// TwinCAT 3 PLC project CassetteLoaderPLC
// ProgramVersion: 3.1.4024.0
// libraries:
//   SPT Base Types, * (Beckhoff Automation LLC)
//   SPT Components, * (Beckhoff Automation LLC)
//   SPT Event Logger, * (Beckhoff Automation LLC)
//   SPT Motion Control, * (Beckhoff Automation LLC)
//   SPT Utilities, * (Beckhoff Automation LLC)
//   Tc2_EtherCAT, * (Beckhoff Automation GmbH)
//   Tc2_Standard, * (Beckhoff Automation GmbH)
//   Tc2_System, * (Beckhoff Automation GmbH)
//   Tc3_EventLogger, * (Beckhoff Automation GmbH)
//   Tc3_Module, * (Beckhoff Automation GmbH)
//   Tc3_PackML_V2, * (Beckhoff Automation GmbH)
//   VisuDialogs, * (System)
//   VisuSymbols, * (System)
// project tree:
//   DUTs/Recipes/ ST_ElevatorRecipe.TcDUT, ST_LoaderRecipe.TcDUT, ST_ShuttleRecipe.TcDUT
//   DUTs/ ST_CassetteStatus.TcDUT, ST_PackML_Control.TcDUT, ST_PackML_Control_Simplified.TcDUT (not stored)
//   / GlobalTextList.TcGTLO, PlcTask.TcTTO, Visualization Manager.TcVMO (not stored)
//   Machine/EquipmentModules/ FB_CassetteLoader.TcPOU
//   Machine/ FB_Machine.TcPOU
//   Machine/HMI Connections/ FB_ControlSource_HMI.TcPOU, FB_ControlSource_HMI_Machine.TcPOU
//   Machine/Templates/ FB_EquipmentModuleTemplate.TcPOU
//   POUs/ MAIN.TcPOU
//   VISUs/VisuOjects/ V_MachineModule.TcVIS, V_Module.TcVIS
//   VISUs/ V_Main.TcVIS
// real-time tasks:
//   TASK PlcTask: cycle T#10ms, priority 20, ADS port 350
// motion (NC):
//   TASK NC-Task 1 SAF: cycle T#2ms, priority 4, ADS port 501
//   TASK NC-Task 1 SVB: cycle T#10ms, priority 8, ADS port 511
//   AXIS Axis-CassetteA (id 1)
//     Dynamic: Acceleration=607.875, Deceleration=607.875, Jerk=1823.62
//     Velo: RefSearch=4.0525, RefSync=4.0525, SlowManual=5, FastManual=50, Fast=405.25, Maximum=405.25
//     OtherSettings: AllowMotionCmdToSlave=true
//     encoder EncType=19
//       EncPara: ScaleFactorNumerator=5, ScaleFactorDenominator=1048576, MaxCount=#xffffffff
//     drive DrvType=16
//       DrvPara: MaxCount=#xffffffff, DriveControlDWord=#x00020000
//         Analog: VeloReferenz=445.775, VeloScale=32, TorqueSetpointScale=10, ScaleFactorActTorque=0.1
//         TimeComp: TaskDelayCycles=1
//     controller CtrType=1
//       CtrPara: PriorControlFactor=1
//         Observer: BandWidth=20
//   AXIS Axis-CassetteB (id 2)
//     Dynamic: Acceleration=607.875, Deceleration=607.875, Jerk=1823.62
//     Velo: RefSearch=4.0525, RefSync=4.0525, SlowManual=5, FastManual=50, Fast=405.25, Maximum=405.25
//     OtherSettings: AllowMotionCmdToSlave=true
//     encoder EncType=19
//       EncPara: ScaleFactorNumerator=5, ScaleFactorDenominator=1048576, MaxCount=#xffffffff
//     drive DrvType=16
//       DrvPara: MaxCount=#xffffffff, DriveControlDWord=#x00020000
//         Analog: VeloReferenz=445.775, VeloScale=32, TorqueSetpointScale=10, ScaleFactorActTorque=0.1
//         TimeComp: TaskDelayCycles=1
//     controller CtrType=1
//       CtrPara: PriorControlFactor=1
//         Observer: BandWidth=20
//   AXIS Axis-Shuttle (id 3)
//     Dynamic: Acceleration=607.875, Deceleration=607.875, Jerk=1823.62
//     Velo: RefSearch=4.0525, RefSync=4.0525, SlowManual=5, FastManual=50, Fast=405.25, Maximum=405.25
//     OtherSettings: AllowMotionCmdToSlave=true
//     encoder EncType=19
//       EncPara: ScaleFactorNumerator=5, ScaleFactorDenominator=1048576, MaxCount=#xffffffff
//     drive DrvType=16
//       DrvPara: MaxCount=#xffffffff, DriveControlDWord=#x00020000
//         Analog: VeloReferenz=445.775, VeloScale=32, TorqueSetpointScale=10, ScaleFactorActTorque=0.1
//         TimeComp: TaskDelayCycles=1
//     controller CtrType=1
//       CtrPara: PriorControlFactor=1
//         Observer: BandWidth=20
// I/O:
//   DEVICE Device 2 (EtherCAT), AmsNetId 169.254.242.100.3.1
//     Term 1 (EK1100) [EK1100 EtherCAT Coupler (2A E-Bus)]
//       Term 2 (EL1098) [EL1098 8Ch. Dig. Input 24V, 10µs, negative]
//       Term 3 (EL7201-9014) [EL7201-9014 1Ch. MDP742 Servo motor output stage with OCT (50V, 2.8A RMS) and STO input]
//       Term 4 (EL7201-9014) [EL7201-9014 1Ch. MDP742 Servo motor output stage with OCT (50V, 2.8A RMS) and STO input]
//       Term 5 (EL7201-9014) [EL7201-9014 1Ch. MDP742 Servo motor output stage with OCT (50V, 2.8A RMS) and STO input]
//       Term 6 (EL2904) [EL2904, 4 Ch. Safety Output 24V, 0.5A, TwinSAFE]
//         modules: Module 1 (FSOES), Module 2 (DO)
//       Term 7 (EL1918) [EL1918, 8Ch. Safety Input 24V, TwinSAFE]
//         modules: Module 1 (FSOE), Module 2 (FSLOGIC)
//       Term 8 (EL9011) [EL9011 End Terminal]
// variable links:
//   NC-Task 1 SAF/Axes/Axis-CassetteA <-> Device 2 (EtherCAT)/Term 1 (EK1100)/Term 3 (EL7201-9014)
//     Drive/Inputs/In/nDcOutputTime <-> InfoData/DcOutputShift
//     Drive/Inputs/In/nState1 <-> DRV Statusword/Statusword
//     Drive/Inputs/In/nState2 <-> DRV Statusword/Statusword @bit 8
//     Drive/Inputs/In/nState4 @bit 1 <-> WcState/InputToggle
//     Drive/Inputs/In/nState4 <-> WcState/WcState
//     Drive/Outputs/Out/nCtrl1 <-> DRV Controlword/Controlword
//     Drive/Outputs/Out/nCtrl2 <-> DRV Controlword/Controlword @bit 8
//     Drive/Outputs/Out/nDataOut2 <-> DRV Target velocity/Target velocity
//     Enc/Inputs/In/nDataIn1 <-> FB Position/Position
//     Enc/Inputs/In/nDcInputTime <-> InfoData/DcInputShift
//     Enc/Inputs/In/nState4 @bit 1 <-> WcState/InputToggle
//     Enc/Inputs/In/nState4 <-> WcState/WcState
//   NC-Task 1 SAF/Axes/Axis-CassetteB <-> Device 2 (EtherCAT)/Term 1 (EK1100)/Term 4 (EL7201-9014)
//     Drive/Inputs/In/nDcOutputTime <-> InfoData/DcOutputShift
//     Drive/Inputs/In/nState1 <-> DRV Statusword/Statusword
//     Drive/Inputs/In/nState2 <-> DRV Statusword/Statusword @bit 8
//     Drive/Inputs/In/nState4 @bit 1 <-> WcState/InputToggle
//     Drive/Inputs/In/nState4 <-> WcState/WcState
//     Drive/Outputs/Out/nCtrl1 <-> DRV Controlword/Controlword
//     Drive/Outputs/Out/nCtrl2 <-> DRV Controlword/Controlword @bit 8
//     Drive/Outputs/Out/nDataOut2 <-> DRV Target velocity/Target velocity
//     Enc/Inputs/In/nDataIn1 <-> FB Position/Position
//     Enc/Inputs/In/nDcInputTime <-> InfoData/DcInputShift
//     Enc/Inputs/In/nState4 @bit 1 <-> WcState/InputToggle
//     Enc/Inputs/In/nState4 <-> WcState/WcState
//   NC-Task 1 SAF/Axes/Axis-Shuttle <-> Device 2 (EtherCAT)/Term 1 (EK1100)/Term 5 (EL7201-9014)
//     Drive/Inputs/In/nDcOutputTime <-> InfoData/DcOutputShift
//     Drive/Inputs/In/nState1 <-> DRV Statusword/Statusword
//     Drive/Inputs/In/nState2 <-> DRV Statusword/Statusword @bit 8
//     Drive/Inputs/In/nState4 @bit 1 <-> WcState/InputToggle
//     Drive/Inputs/In/nState4 <-> WcState/WcState
//     Drive/Outputs/Out/nCtrl1 <-> DRV Controlword/Controlword
//     Drive/Outputs/Out/nCtrl2 <-> DRV Controlword/Controlword @bit 8
//     Drive/Outputs/Out/nDataOut2 <-> DRV Target velocity/Target velocity
//     Enc/Inputs/In/nDataIn1 <-> FB Position/Position
//     Enc/Inputs/In/nDcInputTime <-> InfoData/DcInputShift
//     Enc/Inputs/In/nState4 @bit 1 <-> WcState/InputToggle
//     Enc/Inputs/In/nState4 <-> WcState/WcState
//   CassetteLoaderPLC/CassetteLoaderPLC Instance <-> NC-Task 1 SAF/Axes/Axis-CassetteA
//     PlcTask Inputs/MAIN.CassetteLoaderMachine.CassetteLoaderEM.ElevatorAxisA.BasicAxis._Axis.NcToPlc <-> Outputs/ToPlc
//     PlcTask Outputs/MAIN.CassetteLoaderMachine.CassetteLoaderEM.ElevatorAxisA.BasicAxis._Axis.PlcToNc <-> Inputs/FromPlc
//   CassetteLoaderPLC/CassetteLoaderPLC Instance <-> NC-Task 1 SAF/Axes/Axis-CassetteB
//     PlcTask Inputs/MAIN.CassetteLoaderMachine.CassetteLoaderEM.ElevatorAxisB.BasicAxis._Axis.NcToPlc <-> Outputs/ToPlc
//     PlcTask Outputs/MAIN.CassetteLoaderMachine.CassetteLoaderEM.ElevatorAxisB.BasicAxis._Axis.PlcToNc <-> Inputs/FromPlc
//   CassetteLoaderPLC/CassetteLoaderPLC Instance <-> NC-Task 1 SAF/Axes/Axis-Shuttle
//     PlcTask Inputs/MAIN.CassetteLoaderMachine.CassetteLoaderEM.ShuttleAxis.BasicAxis._Axis.NcToPlc <-> Outputs/ToPlc
//     PlcTask Outputs/MAIN.CassetteLoaderMachine.CassetteLoaderEM.ShuttleAxis.BasicAxis._Axis.PlcToNc <-> Inputs/FromPlc

CONFIGURATION CassetteLoaderPLC
    RESOURCE PLC ON TwinCAT3
        TASK PlcTask(INTERVAL := T#10ms, PRIORITY := 20);
        PROGRAM MAIN WITH PlcTask : MAIN;
    END_RESOURCE
END_CONFIGURATION

// ---- DUTs/Recipes/ST_ElevatorRecipe.TcDUT
TYPE ST_ElevatorRecipe :
STRUCT
	    Velocity     : LREAL;
        Acceleration : LREAL;
		FirstWaveguidePosition : LREAL;
		CassettePitch : LREAL;
		CassetteSlotHeight : LREAL;
		CassetteSlotNumber : INT;
		WaveguideThickness : LREAL;
		BladeThickness : LREAL;
END_STRUCT
END_TYPE

// ---- DUTs/Recipes/ST_LoaderRecipe.TcDUT
TYPE ST_LoaderRecipe :
STRUCT
	    Elevator         		: ST_ElevatorRecipe;
        Shuttle              	: ST_ShuttleRecipe;
END_STRUCT
END_TYPE

// ---- DUTs/Recipes/ST_ShuttleRecipe.TcDUT
TYPE ST_ShuttleRecipe :
STRUCT
		Velocity     : LREAL;
        Acceleration : LREAL;
		CassettePosition : LREAL;
		ToolPosition : LREAL;
END_STRUCT
END_TYPE

// ---- DUTs/ST_CassetteStatus.TcDUT
TYPE ST_CassetteStatus :
STRUCT
	CassetteOnPedestal : BOOL;
	CassetteFull : BOOL;
	CassetteEmpty : BOOL;
	WaveguidePresent : ARRAY[0..23] OF BOOL := [24(FALSE)]; //initiallize none present
	ClearBelowWaveguide : ARRAY[0..23] OF BOOL := [24(FALSE)]; //initiallize not clear
END_STRUCT
END_TYPE

// ---- DUTs/ST_PackML_Control.TcDUT
TYPE ST_PackML_Control :
    STRUCT
        CurrentMode  : E_PMLUnitMode;
        ModeCommand  : E_PMLUnitMode;
        CurrentState : E_PMLState;
        StateCommand : E_PMLCommand;
        ModeNames    : ARRAY[0..31] OF STRING;
    END_STRUCT
END_TYPE

// ---- POUs/MAIN.TcPOU
PROGRAM MAIN
VAR
	ControlSource_HMI : FB_ControlSource_HMI_Machine;
    CassetteLoaderMachine          : FB_Machine := (Name := 'CassetteLoader');
    InitComplete      : BOOL;
END_VAR

CyclicLogic();

METHOD CyclicLogic
VAR_INPUT
END_VAR
IF NOT InitComplete THEN
    InitComplete := Initialize();
    RETURN;
END_IF

//Machine support HMI & Production Monitor
ControlSource_HMI.CyclicLogic();

//Machine Cyclic Logic
CassetteLoaderMachine.CyclicLogic();
END_METHOD

METHOD Initialize : BOOL
VAR_INPUT
END_VAR
//Top level machine initialization should happen here, in the main initialization method. Each subsequent "layer" of modules will be named within their respective "parent" intialize method
_AppInfo.KeepOutputsOnBP := TRUE;
IF NOT ControlSource_HMI.Registered THEN
    CassetteLoaderMachine.RegisterExternalController(ControlSource_HMI);
END_IF

ControlSource_HMI.CyclicLogic();
Initialize := TRUE;
END_METHOD

END_PROGRAM

// ---- Machine/HMI Connections/FB_ControlSource_HMI_Machine.TcPOU
FUNCTION_BLOCK FB_ControlSource_HMI_Machine EXTENDS FB_ControlSource_HMI
VAR_INPUT
END_VAR
VAR_OUTPUT
END_VAR
VAR
END_VAR

METHOD CyclicLogic
VAR_INPUT
END_VAR
SUPER^.CyclicLogic();

//Change the start permissive for the Machine 
MainPMLControl_Simplified.StartPermissive :=
    MainPMLControl_Standard.CurrentState = Tc3_PackML_V2.E_PMLState.ePMLState_Idle OR
    (MainPMLControl_Standard.CurrentState = Tc3_PackML_V2.E_PMLState.ePMLState_Held AND
    MAIN.CassetteLoaderMachine.CurrentState = E_PMLState.ePMLState_Idle);
END_METHOD

END_FUNCTION_BLOCK

// ---- Machine/HMI Connections/FB_ControlSource_HMI.TcPOU
FUNCTION_BLOCK FB_ControlSource_HMI EXTENDS FB_CyclicFB IMPLEMENTS I_PackML_ExternalController
VAR_INPUT
END_VAR

VAR_OUTPUT
END_VAR

VAR
    ipModule                  : I_PackML_Control;
    MainPMLControl_Simplified : ST_PackML_Control_Simplified;
    MainPMLControl_Standard   : ST_PackML_Control;
    R_HMICommand              : R_TRIG;
END_VAR

PROPERTY Control : SPT_BaseTypes.I_PackML_Control
SET
ipModule := Control;
END_SET
END_PROPERTY

METHOD CyclicLogic
VAR
    i : UDINT;
END_VAR
IF NOT _InitComplete THEN
    _InitComplete := Initialize();
    RETURN;
END_IF

MainPMLControl_Standard.CurrentMode  := ipModule.CurrentMode;
MainPMLControl_Standard.CurrentState := ipModule.CurrentState;
FOR i := 1 TO 5 DO
    MainPMLControl_Standard.ModeNames[i] := F_UnitModeToString(UDINT_TO_DINT(i));
END_FOR

//Process HMI requests
R_HMICommand(CLK := (MainPMLControl_Simplified.ResetPressed XOR MainPMLControl_Simplified.StartPressed XOR
                    MainPMLControl_Simplified.StopPressed) XOR
                    (MainPMLControl_Standard.StateCommand <> E_PMLCommand.ePMLCommand_Undefined AND
                    ipModule.StateCommand <> MainPMLControl_Standard.StateCommand) XOR
                    (ipModule.ModeCommand <> MainPMLControl_Standard.ModeCommand));

IF R_HMICommand.Q THEN
    IF MainPMLControl_Simplified.ResetPressed AND MainPMLControl_Simplified.ResetPermissive AND
       MainPMLControl_Standard.CurrentState = E_PMLState.ePMLState_Aborted THEN
        ipModule.ChangeState(Tc3_PackML_V2.E_PMLCommand.ePMLCommand_Clear);
    ELSIF MainPMLControl_Simplified.ResetPressed AND MainPMLControl_Simplified.ResetPermissive THEN
        ipModule.ChangeState(Tc3_PackML_V2.E_PMLCommand.ePMLCommand_Reset);
    ELSIF MainPMLControl_Simplified.StartPressed AND MainPMLControl_Simplified.StartPermissive THEN
        IF MainPMLControl_Standard.CurrentState = Tc3_PackML_V2.E_PMLState.ePMLState_Idle THEN
            ipModule.ChangeState(Tc3_PackML_V2.E_PMLCommand.ePMLCommand_Start);
        ELSIF MainPMLControl_Standard.CurrentState = Tc3_PackML_V2.E_PMLState.ePMLState_Held THEN
            ipModule.ChangeState(Tc3_PackML_V2.E_PMLCommand.ePMLCommand_Unhold);
        END_IF
    ELSIF MainPMLControl_Simplified.StopPressed AND MainPMLControl_Simplified.StopPermissive THEN
        ipModule.ChangeState(Tc3_PackML_V2.E_PMLCommand.ePMLCommand_Stop);
    ELSIF ipModule.StateCommand <> MainPMLControl_Standard.StateCommand THEN
        ipModule.StateCommand := MainPMLControl_Standard.StateCommand;
    ELSIF ipModule.ModeCommand <> MainPMLControl_Standard.ModeCommand THEN
        ipModule.ModeCommand := MainPMLControl_Standard.ModeCommand;
    END_IF
END_IF

MainPMLControl_Simplified.StartPermissive :=
    MainPMLControl_Standard.CurrentState = Tc3_PackML_V2.E_PMLState.ePMLState_Idle OR
    MainPMLControl_Standard.CurrentState = Tc3_PackML_V2.E_PMLState.ePMLState_Held;

MainPMLControl_Simplified.StopPermissive :=
    (MainPMLControl_Standard.CurrentState <> Tc3_PackML_V2.E_PMLState.ePMLState_Stopped AND
     MainPMLControl_Standard.CurrentState <> Tc3_PackML_V2.E_PMLState.ePMLState_Clearing AND
     MainPMLControl_Standard.CurrentState <> Tc3_PackML_V2.E_PMLState.ePMLState_Aborted AND
     MainPMLControl_Standard.CurrentState <> Tc3_PackML_V2.E_PMLState.ePMLState_Aborting AND
     MainPMLControl_Standard.CurrentState <> Tc3_PackML_V2.E_PMLState.ePMLState_Undefined);

MainPMLControl_Simplified.ResetPermissive :=
    MainPMLControl_Standard.CurrentState = Tc3_PackML_V2.E_PMLState.ePMLState_Complete OR
    MainPMLControl_Standard.CurrentState = Tc3_PackML_V2.E_PMLState.ePMLState_Stopped OR
    MainPMLControl_Standard.CurrentState = Tc3_PackML_V2.E_PMLState.ePMLState_Aborted;
END_METHOD

METHOD FINAL Initialize : BOOL
IF Registered THEN
    Initialize := TRUE;
END_IF
END_METHOD

METHOD FINAL ModeChanged
VAR_INPUT
    NewMode : SPT_BaseTypes.E_PMLUnitMode;
END_VAR
MainPMLControl_Standard.ModeCommand := NewMode;
END_METHOD

PROPERTY Registered : BOOL
GET
Registered := ipModule <> 0;
END_GET
END_PROPERTY

METHOD FINAL StateChanged
VAR_INPUT
    NewState : SPT_BaseTypes.E_PMLCommand;
END_VAR
MainPMLControl_Standard.StateCommand := NewState;
END_METHOD

END_FUNCTION_BLOCK

// ---- Machine/FB_Machine.TcPOU
FUNCTION_BLOCK FB_Machine EXTENDS FB_PackML_BaseModule
VAR_INPUT
END_VAR
VAR_OUTPUT
END_VAR
VAR
	//Sub Module 
	CassetteLoaderEM : FB_CassetteLoader := (Name := 'Cassette Loader', LogStateChanges := TRUE); 
	
	// Components

    //Initial List of Components
    ipComponents_Init : ARRAY[1..Parameters_PackML_Base.MAX_NO_OF_COMPONENTS] OF I_ComponentBase := [];

    //Alarms for this module
    MachineAlarms : ARRAY[1..MACHINE_ALARM_COUNT] OF FB_TcAlarm;

	
	//Current Recipe Name
	CurrentRecipeName : STRING;

    //Get Data From PackML? Else RecipeManager is running
    DataFromPackML : BOOL := TRUE;
	
	 //Pack Tags for System
    {attribute 'OPC.UA.DA' := '1'}
    _PackTags : ST_PackMLv30Ext; //ST_PackMLv30 is obsolete in Tc3_PackML_V2
	
END_VAR

// Simulation variables
VAR
    EstopInput  : BOOL;
    LowAirInput : BOOL;
    ErrorInput  : BOOL;
    WarnInput   : BOOL;
    InfoInput   : BOOL;
	ToolLoadUnloadComplete : BOOL;
END_VAR

VAR CONSTANT
    //PackTag parameter IDs
//    LENGTH         : INT := 1;
//    SEALTEMP       : INT := 2;
//    SEALTIME       : INT := 3;
//    PULLWHEELS_VEL : INT := 4;
//    PULLWHEELS_ACC : INT := 5;
//    SEALER_VEL     : INT := 6;
//    SEALER_ACC     : INT := 7;
//    UNWIND_VEL     : INT := 8;
//    UNWIND_ACC     : INT := 9;
//    OPEN_POS       : INT := 10;
//    CLOSED_POS     : INT := 11;

	//Alarm count constant
    MACHINE_ALARM_COUNT : INT := 6;
END_VAR

METHOD PROTECTED Completing
VAR_INPUT
END_VAR
CASE _CurrentMode OF
    //=================================PRODUCTION MODE==================================
    E_PMLUnitMode.ePMLUnitMode_Production:
        StateComplete();
    E_PMLUnitMode.ePMLUnitMode_Maintenance, E_PMLUnitMode.ePMLUnitMode_Manual:
        SUPER^.Completing();
END_CASE
END_METHOD

METHOD PROTECTED CreateEvents
VAR_INPUT
END_VAR
// Add your event creation here
//F_CreateAllEventsInClass(Alarms     := MachineAlarms,
//                         ClassSize  := SIZEOF(TC_Events.VFFSDemo),
//                         pInitEvent := ADR(TC_EVENTS.VFFSDemo.InitReferenceEvent),
//                         Prefix     := Name);

// Super call to base
SUPER^.CreateEvents();
END_METHOD

METHOD CyclicLogic
VAR_INPUT
END_VAR
IF NOT _InitComplete THEN
    _InitComplete := Initialize();
    RETURN;
END_IF

SUPER^.CyclicLogic();

// Fill in the PackTags for the machine output
_PackTags.Status.StateCurrent    := _CurrentState;
_PackTags.Status.UnitModeCurrent := _CurrentMode;

UpdateModeTimers();
END_METHOD

METHOD PROTECTED FINAL Execute
VAR_INPUT
END_VAR
CASE _CurrentMode OF
    //=================================PRODUCTION MODE==================================
    E_PMLUnitMode.ePMLUnitMode_Production:
        (* Run the sequence to make products 
		 Unwind Runs Slowly 
		 Pull Wheels Run 
		 Jaws Seal, and Repeat until production reached*)
//        sealTrig(CLK := SequenceState = 10);
//        IF sealTrig.Q THEN
//            partTimeStart := F_GetActualDcTime64();
//            sealTimeStart := partTimeStart;
//        END_IF

//        pulltrig(CLK := SequenceState = 20);
//        IF pulltrig.Q THEN
//            pullTimeStart := F_GetActualDcTime64();
//        END_IF

//		IF THIS^.Sealer.sealbar.InTempRange THEN
//			CASE SequenceState OF
//				0: //Started
//					Unwind.ChangeState(E_PMLCommand.ePMLCommand_Start);
//					IF Unwind.CurrentState = E_PMLState.ePMLState_Execute THEN
//						SequenceState := SequenceState + 10;
//					END_IF
//				10: // SEAL First
//					Sealer.ChangeState(E_PMLCommand.ePMLCommand_Start);
//					IF Sealer.CurrentState = E_PMLState.ePMLState_Complete THEN
//						Sealer.ChangeState(E_PMLCommand.ePMLCommand_Reset);
//						SequenceState := SequenceState + 10;
//						SealTimeEnd   := F_GetActualDcTime64();
//						sealingTime   := ULINT_TO_LREAL(sealtimeEnd - sealTimeStart) * 1E-9;
//					END_IF
//				20: // Run Pullwheels
//					PullWheels.ChangeState(E_PMLCommand.ePMLCommand_Start);
//					IF PullWheels.CurrentState = E_PMLState.ePMLState_Complete THEN
//						partTimeEnd   := F_GetActualDcTime64();
//						parts         := parts + 1;
//						SequenceState := 10;
//						PullWheels.ChangeState(E_PMLCommand.ePMLCommand_Reset);
//						pullTimeEnd := F_GetActualDcTime64();
//						pullingTime := ULINT_TO_LREAL(pullTimeEnd - pullTimeStart) * 1E-9;
//					END_IF
//			END_CASE
//		ELSE
//			ChangeState(E_PMLCommand.ePMLCommand_Suspend);
//		END_IF
			
    //=================================MAINTENANCE MODE==================================	
    E_PMLUnitMode.ePMLUnitMode_Maintenance:
        ;

    //=================================MANUAL MODE==================================
    E_PMLUnitMode.ePMLUnitMode_Manual:
        ;
END_CASE
END_METHOD

METHOD PROTECTED HMIPermissions
VAR_INPUT
END_VAR
//General Mode Based Monitoring and handling of HMI control
CASE _CurrentMode OF
    E_PMLUnitMode.ePMLUnitMode_Production:
        CASE _CurrentState OF
            E_PMLState.ePMLState_Stopped:
                AllowHMIControl(ThisModuleOnly := TRUE); //Allow control for recovery
            E_PMLState.ePMLState_Idle:
                //BlockHMIControl();
				AllowHMIControl(ThisModuleOnly := TRUE); //Allow control for recovery
            E_PMLState.ePMLState_Suspended:
                BlockHMIControl();
            E_PMLState.ePMLState_Execute:
                BlockHMIControl();
            E_PMLState.ePMLState_Aborted:
                AllowHMIControl(ThisModuleOnly := TRUE); //Allow control for recovery
            E_PMLState.ePMLState_Held:
                AllowHMIControl(ThisModuleOnly := TRUE); //Allow control for recovery
            E_PMLState.ePMLState_Complete:
                BlockHMIControl();
        END_CASE
		
        //AllowHMIControl(ThisModuleOnly := FALSE);
    E_PMLUnitMode.ePMLUnitMode_Manual:
        AllowHMIControl(ThisModuleOnly := FALSE);
    E_PMLUnitMode.ePMLUnitMode_Maintenance:
        AllowHMIControl(ThisModuleOnly := FALSE);
END_CASE
END_METHOD

METHOD PROTECTED Holding
VAR_INPUT
END_VAR
CASE _CurrentMode OF
    //=================================PRODUCTION MODE==================================
    E_PMLUnitMode.ePMLUnitMode_Production:
        IF (CassetteLoaderEM.CurrentState = E_PMLState.ePMLState_Complete OR CassetteLoaderEM.CurrentState = E_PMLState.ePMLState_Idle) THEN
            StateComplete();
        END_IF
    E_PMLUnitMode.ePMLUnitMode_Maintenance, E_PMLUnitMode.ePMLUnitMode_Manual:
        SUPER^.Holding();
	
END_CASE
END_METHOD

METHOD PROTECTED Initialize : BOOL
VAR
    i : UDINT; //Generic iteration value
END_VAR
Initialize := FALSE;
CASE DescendantSequenceState OF
    0:
		RegisterSubmodule(CassetteLoaderEM);

		
        _LogModeChanges         := FALSE;
        _LogStateChanges        := FALSE;
        DescendantSequenceState := DescendantSequenceState + 10;
    10:
        //Setup Custom modes here

        CustomModes(eMode                          :=,
                    sName                          := 'Name',
                    bDisableClearing               := FALSE,
                    bDisableStarting               := FALSE,
                    bDisableSuspended              := FALSE,
                    bDisableStopping               := FALSE,
                    bDisableAborting               := FALSE,
                    bDisableHolding                := TRUE,
                    bDisableHeld                   := TRUE,
                    bDisableUnholding              := TRUE,
                    bDisableSuspending             := FALSE,
                    bDisableUnsuspending           := FALSE,
                    bDisableResetting              := FALSE,
                    bDisableIdle                   := FALSE,
                    bDisableCompleting             := FALSE,
                    bDisableComplete               := FALSE,
                    bEnableUnitModeChangeStopped   := TRUE,
                    bEnableUnitModeChangeIdle      := TRUE,
                    bEnableUnitModeChangeSuspended := FALSE,
                    bEnableUnitModeChangeExecute   := FALSE,
                    bEnableUnitModeChangeAborted   := FALSE,
                    bEnableUnitModeChangeHeld      := FALSE,
                    bEnableUnitModeChangeComplete  := FALSE,
                    bError                         =>,
                    nErrorId                       =>);
        DescendantSequenceState := DescendantSequenceState + 10;
    20:
        //Copy Mode names
        FOR i := 1 TO 3 DO
            ModeNames[i] := F_UnitModeToString(UDINT_TO_DINT(i));
        END_FOR

        DescendantSequenceState := DescendantSequenceState + 10;
    30:
        // Initialize Recipes 
        //Initialize_Recipes();
        DescendantSequenceState := DescendantSequenceState + 10;
    40:
        //Call the Super
        IF SUPER^.Initialize() THEN
            DescendantSequenceState := DescendantSequenceState + 10;
        END_IF
    50:
        Initialize := TRUE;
END_CASE
END_METHOD

METHOD Initialize_Recipes
VAR_INPUT
END_VAR
//// configuration of parameters Max Speed
//_packTags.Command.Parameter[1].ID    := 1;
//_packTags.Command.Parameter[1].Name  := 'Max Speed';
//_packTags.Command.Parameter[1].Unit  := '/min';
//_packTags.Command.Parameter[1].Value := 180;
//_packTags.Command.Parameter[2].ID    := 2;
//_packTags.Command.Parameter[2].Name  := 'Product to Run';
//_packTags.Command.Parameter[2].Unit  := '';
//_packTags.Command.Parameter[2].Value := 1;

//// Recipe Product 1
//_PackTags.Command.Product[1].ProductID                              := 100;
//_PackTags.Command.Product[1].Ingredients[1].IngredientID            := 1;
//_PackTags.Command.Product[1].Ingredients[1].Parameter[1].ID         := _PackTags.Command.Product[1].ProductID * 10 + 1;
//_PackTags.Command.Product[1].Ingredients[1].Parameter[1].Name       := 'Material Type';
//_PackTags.Command.Product[1].Ingredients[1].Parameter[1].Unit       := 'n/a';
//_PackTags.Command.Product[1].Ingredients[1].Parameter[1].Value      := 5;
//_PackTags.Command.Product[1].Ingredients[1].Parameter[2].ID         := _PackTags.Command.Product[1].ProductID * 10 + 2;
//_PackTags.Command.Product[1].Ingredients[1].Parameter[2].Name       := 'Material Thickness';
//_PackTags.Command.Product[1].Ingredients[1].Parameter[2].Unit       := 'um';
//_PackTags.Command.Product[1].Ingredients[1].Parameter[2].Value      := 240;
//_PackTags.Command.Product[1].ProcessVariables[LENGTH].ID            := _PackTags.Command.Product[1].ProductID * 20 + 1;
//_PackTags.Command.Product[1].ProcessVariables[LENGTH].Name          := 'Length';
//_PackTags.Command.Product[1].ProcessVariables[LENGTH].Unit          := 'mm';
//_PackTags.Command.Product[1].ProcessVariables[LENGTH].Value         := 100;
//_PackTags.Command.Product[1].ProcessVariables[SEALTEMP].ID          := _PackTags.Command.Product[1].ProductID * 20 + 2;
//_PackTags.Command.Product[1].ProcessVariables[SEALTEMP].Name        := 'Sealing Temp';
//_PackTags.Command.Product[1].ProcessVariables[SEALTEMP].Unit        := 'C';
//_PackTags.Command.Product[1].ProcessVariables[SEALTEMP].Value       := 100;
//_PackTags.Command.Product[1].ProcessVariables[SEALTIME].ID          := _PackTags.Command.Product[1].ProductID * 20 + 3;
//_PackTags.Command.Product[1].ProcessVariables[SEALTIME].Name        := 'Sealing Time';
//_PackTags.Command.Product[1].ProcessVariables[SEALTIME].Unit        := 'ms';
//_PackTags.Command.Product[1].ProcessVariables[SEALTIME].Value       := 50;
//_PackTags.Command.Product[1].ProcessVariables[PULLWHEELS_VEL].ID    := _PackTags.Command.Product[1].ProductID * 20 + 4;
//_PackTags.Command.Product[1].ProcessVariables[PULLWHEELS_VEL].Name  := 'Pull Wheels Vel';
//_PackTags.Command.Product[1].ProcessVariables[PULLWHEELS_VEL].Unit  := 'mm/s';
//_PackTags.Command.Product[1].ProcessVariables[PULLWHEELS_VEL].Value := 100;
//_PackTags.Command.Product[1].ProcessVariables[PULLWHEELS_ACC].ID    := _PackTags.Command.Product[1].ProductID * 20 + 5;
//_PackTags.Command.Product[1].ProcessVariables[PULLWHEELS_ACC].Name  := 'Pull Wheels Acc';
//_PackTags.Command.Product[1].ProcessVariables[PULLWHEELS_ACC].Unit  := 'mm/s2';
//_PackTags.Command.Product[1].ProcessVariables[PULLWHEELS_ACC].Value := 1000;
//_PackTags.Command.Product[1].ProcessVariables[OPEN_POS].ID          := _PackTags.Command.Product[1].ProductID * 20 + 6;
//_PackTags.Command.Product[1].ProcessVariables[OPEN_POS].Name        := 'Sealer Open Position';
//_PackTags.Command.Product[1].ProcessVariables[OPEN_POS].Unit        := 'mm';
//_PackTags.Command.Product[1].ProcessVariables[OPEN_POS].Value       := 105;
//_PackTags.Command.Product[1].ProcessVariables[CLOSED_POS].ID        := _PackTags.Command.Product[1].ProductID * 20 + 7;
//_PackTags.Command.Product[1].ProcessVariables[CLOSED_POS].Name      := 'Sealer Closed Position';
//_PackTags.Command.Product[1].ProcessVariables[CLOSED_POS].Unit      := 'mm';
//_PackTags.Command.Product[1].ProcessVariables[CLOSED_POS].Value     := 250;
//_PackTags.Command.Product[1].ProcessVariables[SEALER_VEL].ID        := _PackTags.Command.Product[1].ProductID * 20 + 8;
//_PackTags.Command.Product[1].ProcessVariables[SEALER_VEL].Name      := 'Sealer Vel';
//_PackTags.Command.Product[1].ProcessVariables[SEALER_VEL].Unit      := 'mm/s';
//_PackTags.Command.Product[1].ProcessVariables[SEALER_VEL].Value     := 100;
//_PackTags.Command.Product[1].ProcessVariables[SEALER_ACC].ID        := _PackTags.Command.Product[1].ProductID * 20 + 9;
//_PackTags.Command.Product[1].ProcessVariables[SEALER_ACC].Name      := 'Sealer Acc';
//_PackTags.Command.Product[1].ProcessVariables[SEALER_ACC].Unit      := 'mm/s2';
//_PackTags.Command.Product[1].ProcessVariables[SEALER_ACC].Value     := 1000;
//_PackTags.Command.Product[1].ProcessVariables[UNWIND_VEL].ID        := _PackTags.Command.Product[1].ProductID * 20 + 10;
//_PackTags.Command.Product[1].ProcessVariables[UNWIND_VEL].Name      := 'Unwind Vel';
//_PackTags.Command.Product[1].ProcessVariables[UNWIND_VEL].Unit      := 'mm/s';
//_PackTags.Command.Product[1].ProcessVariables[UNWIND_VEL].Value     := 100;
//_PackTags.Command.Product[1].ProcessVariables[UNWIND_ACC].ID        := _PackTags.Command.Product[1].ProductID * 20 + 11;
//_PackTags.Command.Product[1].ProcessVariables[UNWIND_ACC].Name      := 'Unwind Acc';
//_PackTags.Command.Product[1].ProcessVariables[UNWIND_ACC].Unit      := 'mm/s2';
//_PackTags.Command.Product[1].ProcessVariables[UNWIND_ACC].Value     := 1000;

//// Product 2
//_PackTags.Command.Product[2].ProductID                         := 100;
//_PackTags.Command.Product[2].Ingredients[1].IngredientID       := 1;
//_PackTags.Command.Product[2].Ingredients[1].Parameter[1].ID    := _PackTags.Command.Product[1].ProductID * 10 + 1;
//_PackTags.Command.Product[2].Ingredients[1].Parameter[1].Name  := 'Material Type';
//_PackTags.Command.Product[2].Ingredients[1].Parameter[1].Unit  := 'n/a';
//_PackTags.Command.Product[2].Ingredients[1].Parameter[1].Value := 2;
//_PackTags.Command.Product[2].Ingredients[1].Parameter[2].ID    := _PackTags.Command.Product[1].ProductID * 10 + 2;
//_PackTags.Command.Product[2].Ingredients[1].Parameter[2].Name  := 'Material Thickness';
//_PackTags.Command.Product[2].Ingredients[1].Parameter[2].Unit  := 'um';
//_PackTags.Command.Product[2].Ingredients[1].Parameter[2].Value := 220;
//_PackTags.Command.Product[2].ProcessVariables[LENGTH].ID       := _PackTags.Command.Product[1].ProductID * 20 + 1;
//_PackTags.Command.Product[2].ProcessVariables[LENGTH].Name     := 'Length';
//_PackTags.Command.Product[2].ProcessVariables[LENGTH].Unit     := 'mm';
//_PackTags.Command.Product[2].ProcessVariables[LENGTH].Value    := 55;
//_PackTags.Command.Product[2].ProcessVariables[SEALTEMP].ID     := _PackTags.Command.Product[1].ProductID * 20 + 2;
//_PackTags.Command.Product[2].ProcessVariables[SEALTEMP].Name   := 'Sealing Temp';
//_PackTags.Command.Product[2].ProcessVariables[SEALTEMP].Unit   := 'C';
//_PackTags.Command.Product[2].ProcessVariables[SEALTEMP].Value  := 110;
//_PackTags.Command.Product[2].ProcessVariables[SEALTIME].ID     := _PackTags.Command.Product[1].ProductID * 20 + 3;
//_PackTags.Command.Product[2].ProcessVariables[SEALTIME].Name   := 'Sealing Time';
//_PackTags.Command.Product[2].ProcessVariables[SEALTIME].Unit   := 'ms';
//_PackTags.Command.Product[2].ProcessVariables[SEALTIME].Value  := 100;
//_PackTags.Command.Product[2].ProcessVariables[PULLWHEELS_VEL].ID    := _PackTags.Command.Product[1].ProductID * 20 + 4;
//_PackTags.Command.Product[2].ProcessVariables[PULLWHEELS_VEL].Name  := 'Pull Wheels Vel';
//_PackTags.Command.Product[2].ProcessVariables[PULLWHEELS_VEL].Unit  := 'mm/s';
//_PackTags.Command.Product[2].ProcessVariables[PULLWHEELS_VEL].Value := 200;
//_PackTags.Command.Product[2].ProcessVariables[PULLWHEELS_ACC].ID    := _PackTags.Command.Product[1].ProductID * 20 + 5;
//_PackTags.Command.Product[2].ProcessVariables[PULLWHEELS_ACC].Name  := 'Pull Wheels Acc';
//_PackTags.Command.Product[2].ProcessVariables[PULLWHEELS_ACC].Unit  := 'mm/s2';
//_PackTags.Command.Product[2].ProcessVariables[PULLWHEELS_ACC].Value := 2000;
//_PackTags.Command.Product[2].ProcessVariables[OPEN_POS].ID          := _PackTags.Command.Product[1].ProductID * 20 + 6;
//_PackTags.Command.Product[2].ProcessVariables[OPEN_POS].Name        := 'Sealer Open Position';
//_PackTags.Command.Product[2].ProcessVariables[OPEN_POS].Unit        := 'mm';
//_PackTags.Command.Product[2].ProcessVariables[OPEN_POS].Value       := 60;
//_PackTags.Command.Product[2].ProcessVariables[CLOSED_POS].ID        := _PackTags.Command.Product[1].ProductID * 20 + 7;
//_PackTags.Command.Product[2].ProcessVariables[CLOSED_POS].Name      := 'Sealer Closed Position';
//_PackTags.Command.Product[2].ProcessVariables[CLOSED_POS].Unit      := 'mm';
//_PackTags.Command.Product[2].ProcessVariables[CLOSED_POS].Value     := 253;
//_PackTags.Command.Product[2].ProcessVariables[SEALER_VEL].ID        := _PackTags.Command.Product[1].ProductID * 20 + 8;
//_PackTags.Command.Product[2].ProcessVariables[SEALER_VEL].Name      := 'Sealer Vel';
//_PackTags.Command.Product[2].ProcessVariables[SEALER_VEL].Unit      := 'mm/s';
//_PackTags.Command.Product[2].ProcessVariables[SEALER_VEL].Value     := 200;
//_PackTags.Command.Product[2].ProcessVariables[SEALER_ACC].ID        := _PackTags.Command.Product[1].ProductID * 20 + 9;
//_PackTags.Command.Product[2].ProcessVariables[SEALER_ACC].Name      := 'Sealer Acc';
//_PackTags.Command.Product[2].ProcessVariables[SEALER_ACC].Unit      := 'mm/s2';
//_PackTags.Command.Product[2].ProcessVariables[SEALER_ACC].Value     := 2000;
//_PackTags.Command.Product[2].ProcessVariables[UNWIND_VEL].ID        := _PackTags.Command.Product[1].ProductID * 20 + 10;
//_PackTags.Command.Product[2].ProcessVariables[UNWIND_VEL].Name      := 'Unwind Vel';
//_PackTags.Command.Product[2].ProcessVariables[UNWIND_VEL].Unit      := 'mm/s';
//_PackTags.Command.Product[2].ProcessVariables[UNWIND_VEL].Value     := 200;
//_PackTags.Command.Product[2].ProcessVariables[UNWIND_ACC].ID        := _PackTags.Command.Product[1].ProductID * 20 + 11;
//_PackTags.Command.Product[2].ProcessVariables[UNWIND_ACC].Name      := 'Unwind Acc';
//_PackTags.Command.Product[2].ProcessVariables[UNWIND_ACC].Unit      := 'mm/s2';
//_PackTags.Command.Product[2].ProcessVariables[UNWIND_ACC].Value     := 2000;

////Product 3
//_PackTags.Command.Product[3].ProductID                         := 307;
//_PackTags.Command.Product[3].Ingredients[1].IngredientID       := 1;
//_PackTags.Command.Product[3].Ingredients[1].Parameter[1].ID    := _PackTags.Command.Product[1].ProductID * 10 + 1;
//_PackTags.Command.Product[3].Ingredients[1].Parameter[1].Name  := 'Material Type';
//_PackTags.Command.Product[3].Ingredients[1].Parameter[1].Unit  := 'n/a';
//_PackTags.Command.Product[3].Ingredients[1].Parameter[1].Value := 2;
//_PackTags.Command.Product[3].Ingredients[1].Parameter[2].ID    := _PackTags.Command.Product[1].ProductID * 10 + 2;
//_PackTags.Command.Product[3].Ingredients[1].Parameter[2].Name  := 'Material Thickness';
//_PackTags.Command.Product[3].Ingredients[1].Parameter[2].Unit  := 'um';
//_PackTags.Command.Product[3].Ingredients[1].Parameter[2].Value := 220;
//_PackTags.Command.Product[3].ProcessVariables[LENGTH].ID       := _PackTags.Command.Product[1].ProductID * 20 + 1;
//_PackTags.Command.Product[3].ProcessVariables[LENGTH].Name     := 'Length';
//_PackTags.Command.Product[3].ProcessVariables[LENGTH].Unit     := 'mm';
//_PackTags.Command.Product[3].ProcessVariables[LENGTH].Value    := 85;
//_PackTags.Command.Product[3].ProcessVariables[SEALTEMP].ID     := _PackTags.Command.Product[1].ProductID * 20 + 2;
//_PackTags.Command.Product[3].ProcessVariables[SEALTEMP].Name   := 'Sealing Temp';
//_PackTags.Command.Product[3].ProcessVariables[SEALTEMP].Unit   := 'C';
//_PackTags.Command.Product[3].ProcessVariables[SEALTEMP].Value  := 95;
//_PackTags.Command.Product[3].ProcessVariables[SEALTIME].ID     := _PackTags.Command.Product[1].ProductID * 20 + 3;
//_PackTags.Command.Product[3].ProcessVariables[SEALTIME].Name   := 'Sealing Time';
//_PackTags.Command.Product[3].ProcessVariables[SEALTIME].Unit   := 'ms';
//_PackTags.Command.Product[3].ProcessVariables[SEALTIME].Value  := 20;
//_PackTags.Command.Product[3].ProcessVariables[PULLWHEELS_VEL].ID    := _PackTags.Command.Product[1].ProductID * 20 + 4;
//_PackTags.Command.Product[3].ProcessVariables[PULLWHEELS_VEL].Name  := 'Pull Wheels Vel';
//_PackTags.Command.Product[3].ProcessVariables[PULLWHEELS_VEL].Unit  := 'mm/s';
//_PackTags.Command.Product[3].ProcessVariables[PULLWHEELS_VEL].Value := 300;
//_PackTags.Command.Product[3].ProcessVariables[PULLWHEELS_ACC].ID    := _PackTags.Command.Product[1].ProductID * 20 + 5;
//_PackTags.Command.Product[3].ProcessVariables[PULLWHEELS_ACC].Name  := 'Pull Wheels Acc';
//_PackTags.Command.Product[3].ProcessVariables[PULLWHEELS_ACC].Unit  := 'mm/s2';
//_PackTags.Command.Product[3].ProcessVariables[PULLWHEELS_ACC].Value := 3000;
//_PackTags.Command.Product[3].ProcessVariables[OPEN_POS].ID          := _PackTags.Command.Product[1].ProductID * 20 + 6;
//_PackTags.Command.Product[3].ProcessVariables[OPEN_POS].Name        := 'Sealer Open Position';
//_PackTags.Command.Product[3].ProcessVariables[OPEN_POS].Unit        := 'mm';
//_PackTags.Command.Product[3].ProcessVariables[OPEN_POS].Value       := 56;
//_PackTags.Command.Product[3].ProcessVariables[CLOSED_POS].ID        := _PackTags.Command.Product[1].ProductID * 20 + 7;
//_PackTags.Command.Product[3].ProcessVariables[CLOSED_POS].Name      := 'Sealer Closed Position';
//_PackTags.Command.Product[3].ProcessVariables[CLOSED_POS].Unit      := 'mm';
//_PackTags.Command.Product[3].ProcessVariables[CLOSED_POS].Value     := 265;
//_PackTags.Command.Product[3].ProcessVariables[SEALER_VEL].ID        := _PackTags.Command.Product[1].ProductID * 20 + 8;
//_PackTags.Command.Product[3].ProcessVariables[SEALER_VEL].Name      := 'Sealer Vel';
//_PackTags.Command.Product[3].ProcessVariables[SEALER_VEL].Unit      := 'mm/s';
//_PackTags.Command.Product[3].ProcessVariables[SEALER_VEL].Value     := 300;
//_PackTags.Command.Product[3].ProcessVariables[SEALER_ACC].ID        := _PackTags.Command.Product[1].ProductID * 20 + 9;
//_PackTags.Command.Product[3].ProcessVariables[SEALER_ACC].Name      := 'Sealer Acc';
//_PackTags.Command.Product[3].ProcessVariables[SEALER_ACC].Unit      := 'mm/s2';
//_PackTags.Command.Product[3].ProcessVariables[SEALER_ACC].Value     := 3000;
//_PackTags.Command.Product[3].ProcessVariables[UNWIND_VEL].ID        := _PackTags.Command.Product[1].ProductID * 20 + 10;
//_PackTags.Command.Product[3].ProcessVariables[UNWIND_VEL].Name      := 'Unwind Vel';
//_PackTags.Command.Product[3].ProcessVariables[UNWIND_VEL].Unit      := 'mm/s';
//_PackTags.Command.Product[3].ProcessVariables[UNWIND_VEL].Value     := 300;
//_PackTags.Command.Product[3].ProcessVariables[UNWIND_ACC].ID        := _PackTags.Command.Product[1].ProductID * 20 + 11;
//_PackTags.Command.Product[3].ProcessVariables[UNWIND_ACC].Name      := 'Unwind Acc';
//_PackTags.Command.Product[3].ProcessVariables[UNWIND_ACC].Unit      := 'mm/s2';
//_PackTags.Command.Product[3].ProcessVariables[UNWIND_ACC].Value     := 3000;

////Product 4
//_PackTags.Command.Product[4].ProductID                         := 401;
//_PackTags.Command.Product[4].Ingredients[1].IngredientID       := 1;
//_PackTags.Command.Product[4].Ingredients[1].Parameter[1].ID    := _PackTags.Command.Product[1].ProductID * 10 + 1;
//_PackTags.Command.Product[4].Ingredients[1].Parameter[1].Name  := 'Material Type';
//_PackTags.Command.Product[4].Ingredients[1].Parameter[1].Unit  := 'n/a';
//_PackTags.Command.Product[4].Ingredients[1].Parameter[1].Value := 2;
//_PackTags.Command.Product[4].Ingredients[1].Parameter[2].ID    := _PackTags.Command.Product[1].ProductID * 10 + 2;
//_PackTags.Command.Product[4].Ingredients[1].Parameter[2].Name  := 'Material Thickness';
//_PackTags.Command.Product[4].Ingredients[1].Parameter[2].Unit  := 'um';
//_PackTags.Command.Product[4].Ingredients[1].Parameter[2].Value := 220;
//_PackTags.Command.Product[4].ProcessVariables[LENGTH].ID       := _PackTags.Command.Product[1].ProductID * 20 + 1;
//_PackTags.Command.Product[4].ProcessVariables[LENGTH].Name     := 'Length';
//_PackTags.Command.Product[4].ProcessVariables[LENGTH].Unit     := 'mm';
//_PackTags.Command.Product[4].ProcessVariables[LENGTH].Value    := 85;
//_PackTags.Command.Product[4].ProcessVariables[SEALTEMP].ID     := _PackTags.Command.Product[1].ProductID * 20 + 2;
//_PackTags.Command.Product[4].ProcessVariables[SEALTEMP].Name   := 'Sealing Temp';
//_PackTags.Command.Product[4].ProcessVariables[SEALTEMP].Unit   := 'C';
//_PackTags.Command.Product[4].ProcessVariables[SEALTEMP].Value  := 95;
//_PackTags.Command.Product[4].ProcessVariables[SEALTIME].ID     := _PackTags.Command.Product[1].ProductID * 20 + 3;
//_PackTags.Command.Product[4].ProcessVariables[SEALTIME].Name   := 'Sealing Time';
//_PackTags.Command.Product[4].ProcessVariables[SEALTIME].Unit   := 'ms';
//_PackTags.Command.Product[4].ProcessVariables[SEALTIME].Value  := 80;
//_PackTags.Command.Product[4].ProcessVariables[PULLWHEELS_VEL].ID    := _PackTags.Command.Product[1].ProductID * 20 + 4;
//_PackTags.Command.Product[4].ProcessVariables[PULLWHEELS_VEL].Name  := 'Pull Wheels Vel';
//_PackTags.Command.Product[4].ProcessVariables[PULLWHEELS_VEL].Unit  := 'mm/s';
//_PackTags.Command.Product[4].ProcessVariables[PULLWHEELS_VEL].Value := 100;
//_PackTags.Command.Product[4].ProcessVariables[PULLWHEELS_ACC].ID    := _PackTags.Command.Product[1].ProductID * 20 + 5;
//_PackTags.Command.Product[4].ProcessVariables[PULLWHEELS_ACC].Name  := 'Pull Wheels Acc';
//_PackTags.Command.Product[4].ProcessVariables[PULLWHEELS_ACC].Unit  := 'mm/s2';
//_PackTags.Command.Product[4].ProcessVariables[PULLWHEELS_ACC].Value := 1000;
//_PackTags.Command.Product[4].ProcessVariables[OPEN_POS].ID          := _PackTags.Command.Product[1].ProductID * 20 + 6;
//_PackTags.Command.Product[4].ProcessVariables[OPEN_POS].Name        := 'Sealer Open Position';
//_PackTags.Command.Product[4].ProcessVariables[OPEN_POS].Unit        := 'mm';
//_PackTags.Command.Product[4].ProcessVariables[OPEN_POS].Value       := 105;
//_PackTags.Command.Product[4].ProcessVariables[CLOSED_POS].ID        := _PackTags.Command.Product[1].ProductID * 20 + 7;
//_PackTags.Command.Product[4].ProcessVariables[CLOSED_POS].Name      := 'Sealer Closed Position';
//_PackTags.Command.Product[4].ProcessVariables[CLOSED_POS].Unit      := 'mm';
//_PackTags.Command.Product[4].ProcessVariables[CLOSED_POS].Value     := 250;
//_PackTags.Command.Product[4].ProcessVariables[SEALER_VEL].ID        := _PackTags.Command.Product[1].ProductID * 20 + 8;
//_PackTags.Command.Product[4].ProcessVariables[SEALER_VEL].Name      := 'Sealer Vel';
//_PackTags.Command.Product[4].ProcessVariables[SEALER_VEL].Unit      := 'mm/s';
//_PackTags.Command.Product[4].ProcessVariables[SEALER_VEL].Value     := 100;
//_PackTags.Command.Product[4].ProcessVariables[SEALER_ACC].ID        := _PackTags.Command.Product[1].ProductID * 20 + 9;
//_PackTags.Command.Product[4].ProcessVariables[SEALER_ACC].Name      := 'Sealer Acc';
//_PackTags.Command.Product[4].ProcessVariables[SEALER_ACC].Unit      := 'mm/s2';
//_PackTags.Command.Product[4].ProcessVariables[SEALER_ACC].Value     := 1000;
//_PackTags.Command.Product[4].ProcessVariables[UNWIND_VEL].ID        := _PackTags.Command.Product[1].ProductID * 20 + 10;
//_PackTags.Command.Product[4].ProcessVariables[UNWIND_VEL].Name      := 'Unwind Vel';
//_PackTags.Command.Product[4].ProcessVariables[UNWIND_VEL].Unit      := 'mm/s';
//_PackTags.Command.Product[4].ProcessVariables[UNWIND_VEL].Value     := 100;
//_PackTags.Command.Product[4].ProcessVariables[UNWIND_ACC].ID        := _PackTags.Command.Product[1].ProductID * 20 + 11;
//_PackTags.Command.Product[4].ProcessVariables[UNWIND_ACC].Name      := 'Unwind Acc';
//_PackTags.Command.Product[4].ProcessVariables[UNWIND_ACC].Unit      := 'mm/s2';
//_PackTags.Command.Product[4].ProcessVariables[UNWIND_ACC].Value     := 1000;

////Product 5
//_PackTags.Command.Product[5].ProductID                         := 522;
//_PackTags.Command.Product[5].Ingredients[1].IngredientID       := 1;
//_PackTags.Command.Product[5].Ingredients[1].Parameter[1].ID    := _PackTags.Command.Product[1].ProductID * 10 + 1;
//_PackTags.Command.Product[5].Ingredients[1].Parameter[1].Name  := 'Material Type';
//_PackTags.Command.Product[5].Ingredients[1].Parameter[1].Unit  := 'n/a';
//_PackTags.Command.Product[5].Ingredients[1].Parameter[1].Value := 2;
//_PackTags.Command.Product[5].Ingredients[1].Parameter[2].ID    := _PackTags.Command.Product[1].ProductID * 10 + 2;
//_PackTags.Command.Product[5].Ingredients[1].Parameter[2].Name  := 'Material Thickness';
//_PackTags.Command.Product[5].Ingredients[1].Parameter[2].Unit  := 'um';
//_PackTags.Command.Product[5].Ingredients[1].Parameter[2].Value := 520;
//_PackTags.Command.Product[5].ProcessVariables[LENGTH].ID       := _PackTags.Command.Product[1].ProductID * 20 + 1;
//_PackTags.Command.Product[5].ProcessVariables[LENGTH].Name     := 'Length';
//_PackTags.Command.Product[5].ProcessVariables[LENGTH].Unit     := 'mm';
//_PackTags.Command.Product[5].ProcessVariables[LENGTH].Value    := 200;
//_PackTags.Command.Product[5].ProcessVariables[SEALTEMP].ID     := _PackTags.Command.Product[1].ProductID * 20 + 2;
//_PackTags.Command.Product[5].ProcessVariables[SEALTEMP].Name   := 'Sealing Temp';
//_PackTags.Command.Product[5].ProcessVariables[SEALTEMP].Unit   := 'C';
//_PackTags.Command.Product[5].ProcessVariables[SEALTEMP].Value  := 130;
//_PackTags.Command.Product[5].ProcessVariables[SEALTIME].ID     := _PackTags.Command.Product[1].ProductID * 20 + 3;
//_PackTags.Command.Product[5].ProcessVariables[SEALTIME].Name   := 'Sealing Time';
//_PackTags.Command.Product[5].ProcessVariables[SEALTIME].Unit   := 'ms';
//_PackTags.Command.Product[5].ProcessVariables[SEALTIME].Value  := 200;
//_PackTags.Command.Product[5].ProcessVariables[PULLWHEELS_VEL].ID    := _PackTags.Command.Product[1].ProductID * 20 + 4;
//_PackTags.Command.Product[5].ProcessVariables[PULLWHEELS_VEL].Name  := 'Pull Wheels Vel';
//_PackTags.Command.Product[5].ProcessVariables[PULLWHEELS_VEL].Unit  := 'mm/s';
//_PackTags.Command.Product[5].ProcessVariables[PULLWHEELS_VEL].Value := 100;
//_PackTags.Command.Product[5].ProcessVariables[PULLWHEELS_ACC].ID    := _PackTags.Command.Product[1].ProductID * 20 + 5;
//_PackTags.Command.Product[5].ProcessVariables[PULLWHEELS_ACC].Name  := 'Pull Wheels Acc';
//_PackTags.Command.Product[5].ProcessVariables[PULLWHEELS_ACC].Unit  := 'mm/s2';
//_PackTags.Command.Product[5].ProcessVariables[PULLWHEELS_ACC].Value := 1000;
//_PackTags.Command.Product[5].ProcessVariables[OPEN_POS].ID          := _PackTags.Command.Product[1].ProductID * 20 + 6;
//_PackTags.Command.Product[5].ProcessVariables[OPEN_POS].Name        := 'Sealer Open Position';
//_PackTags.Command.Product[5].ProcessVariables[OPEN_POS].Unit        := 'mm';
//_PackTags.Command.Product[5].ProcessVariables[OPEN_POS].Value       := 105;
//_PackTags.Command.Product[5].ProcessVariables[CLOSED_POS].ID        := _PackTags.Command.Product[1].ProductID * 20 + 7;
//_PackTags.Command.Product[5].ProcessVariables[CLOSED_POS].Name      := 'Sealer Closed Position';
//_PackTags.Command.Product[5].ProcessVariables[CLOSED_POS].Unit      := 'mm';
//_PackTags.Command.Product[5].ProcessVariables[CLOSED_POS].Value     := 250;
//_PackTags.Command.Product[5].ProcessVariables[SEALER_VEL].ID        := _PackTags.Command.Product[1].ProductID * 20 + 8;
//_PackTags.Command.Product[5].ProcessVariables[SEALER_VEL].Name      := 'Sealer Vel';
//_PackTags.Command.Product[5].ProcessVariables[SEALER_VEL].Unit      := 'mm/s';
//_PackTags.Command.Product[5].ProcessVariables[SEALER_VEL].Value     := 100;
//_PackTags.Command.Product[5].ProcessVariables[SEALER_ACC].ID        := _PackTags.Command.Product[1].ProductID * 20 + 9;
//_PackTags.Command.Product[5].ProcessVariables[SEALER_ACC].Name      := 'Sealer Acc';
//_PackTags.Command.Product[5].ProcessVariables[SEALER_ACC].Unit      := 'mm/s2';
//_PackTags.Command.Product[5].ProcessVariables[SEALER_ACC].Value     := 1000;
//_PackTags.Command.Product[5].ProcessVariables[UNWIND_VEL].ID        := _PackTags.Command.Product[1].ProductID * 20 + 10;
//_PackTags.Command.Product[5].ProcessVariables[UNWIND_VEL].Name      := 'Unwind Vel';
//_PackTags.Command.Product[5].ProcessVariables[UNWIND_VEL].Unit      := 'mm/s';
//_PackTags.Command.Product[5].ProcessVariables[UNWIND_VEL].Value     := 100;
//_PackTags.Command.Product[5].ProcessVariables[UNWIND_ACC].ID        := _PackTags.Command.Product[1].ProductID * 20 + 11;
//_PackTags.Command.Product[5].ProcessVariables[UNWIND_ACC].Name      := 'Unwind Acc';
//_PackTags.Command.Product[5].ProcessVariables[UNWIND_ACC].Unit      := 'mm/s2';
//_PackTags.Command.Product[5].ProcessVariables[UNWIND_ACC].Value     := 1000;


CurrentRecipeName := 'From PackTags';
END_METHOD

PROPERTY PUBLIC PackTags : ST_PackMLv30Ext
GET
PackTags := _packTags;
END_GET
END_PROPERTY

METHOD RaiseAlarm2Args
VAR_IN_OUT
    Alarm : FB_TcAlarm; //Alarm to be raised
END_VAR

VAR_INPUT
    String_1 : STRING; //First String Parameter (The Name of this component will be applied first automatically)
    String_2 : STRING; //Second String Parameter
END_VAR
F_RaiseAlarmWithStringParameters(Alarm    := Alarm,
                                 String_1 := Name,
                                 String_2 := String_1,
                                 String_3 := String_2);
END_METHOD

METHOD PROTECTED Resetting
VAR_INPUT
END_VAR
CASE _CurrentMode OF
    //=================================PRODUCTION MODE==================================
    E_PMLUnitMode.ePMLUnitMode_Production:
        IF DataFromPackML THEN
//            product           := LREAL_TO_INT(_PackTags.Command.Parameter[2].Value);
//            PullWheels.Length := _PackTags.Command.Product[product].ProcessVariables[LENGTH].Value;
//			PullWheels.Velocity := _PackTags.Command.Product[product].ProcessVariables[PULLWHEELS_VEL].Value;
//			PullWheels.Acceleration := _PackTags.Command.Product[product].ProcessVariables[PULLWHEELS_ACC].Value;
//            Sealer.SealTime   := _PackTags.Command.Product[product].ProcessVariables[SEALTIME].Value;
//            Sealer.Temp       := _PackTags.Command.Product[product].ProcessVariables[SEALTEMP].Value;
//			Sealer.OpenPos := _PackTags.Command.Product[product].ProcessVariables[OPEN_POS].Value;
//			Sealer.ClosedPos := _PackTags.Command.Product[product].ProcessVariables[CLOSED_POS].Value;
//			Sealer.Velocity := _PackTags.Command.Product[product].ProcessVariables[SEALER_VEL].Value;
//			Sealer.Acceleration := _PackTags.Command.Product[product].ProcessVariables[SEALER_ACC].Value;
//			Unwind.Velocity := _PackTags.Command.Product[product].ProcessVariables[UNWIND_VEL].Value;
//			Unwind.Acceleration := _PackTags.Command.Product[product].ProcessVariables[UNWIND_ACC].Value;
        END_IF

    E_PMLUnitMode.ePMLUnitMode_Maintenance, E_PMLUnitMode.ePMLUnitMode_Manual:
        ;
END_CASE

SUPER^.Resetting();
END_METHOD

METHOD PROTECTED Starting
VAR_INPUT
END_VAR
CASE _CurrentMode OF
    //=================================PRODUCTION MODE==================================
    E_PMLUnitMode.ePMLUnitMode_Production:
        // The seal bar can go to Execute, the others will be run in Mahcine Execute
        //Sealer.Heat := TRUE;
        StateComplete();
    E_PMLUnitMode.ePMLUnitMode_Maintenance, E_PMLUnitMode.ePMLUnitMode_Manual:
        SUPER^.Starting();
END_CASE
END_METHOD

METHOD PROTECTED SubModuleMonitor : BOOL
VAR
    AlarmResponses : ARRAY[0..4] OF E_AlarmResponse; //Temporary response array	
END_VAR
// Check the sub Modules for Alarm Severity
SUPER^.SubModuleMonitor();

//Check the alarms at the machine level
_CurrentAlarmSeverity := F_GetMaxSeverityRaised(Alarms := MachineAlarms, CurrentSeverity := _CurrentAlarmSeverity);

//Check the severity of the machine level alarms
IF _CurrentState <> E_PMLState.ePMLState_Aborted AND _CurrentState <> E_PMLState.ePMLState_Aborting AND _CurrentState <> E_PMLState.ePMLState_Clearing AND
   _CurrentState <> E_PMLState.ePMLState_Stopped AND _CurrentState <> E_PMLState.ePMLState_Stopping THEN
    AlarmResponses := _ParentFaultResponseDefinitions;
    CASE AlarmResponses[CurrentAlarmSeverity] OF
        E_AlarmResponse.Abort_ImmediateError:
            AbortImmediateError(Name, TRUE);
        E_AlarmResponse.Abort_Immediate:
            AbortImmediate();
        E_AlarmResponse.Stop_Immediate:
            StopImmediate();
        E_AlarmResponse.Stop_Controlled:
            StopControlled();
        E_AlarmResponse.Hold_Immediate:
            HoldImmediate();
        E_AlarmResponse.Suspend_Immediate:
            SuspendImmediate();
        E_AlarmResponse.Suspend_Controlled:
            SuspendControlled();
        E_AlarmResponse.NoResponse:
            ;
    END_CASE
ELSIF _CurrentState = E_PMLState.ePMLState_Stopped OR _CurrentState = E_PMLState.ePMLState_Stopping THEN
    AlarmResponses := _ParentFaultResponseDefinitions;
    CASE AlarmResponses[CurrentAlarmSeverity] OF
        E_AlarmResponse.Abort_ImmediateError:
            AbortImmediateError(Name, TRUE);
        E_AlarmResponse.Abort_Immediate:
            AbortImmediate();
        E_AlarmResponse.NoResponse:
            ;
    END_CASE
END_IF
END_METHOD

METHOD PROTECTED Suspended
VAR_INPUT
END_VAR

//wait for the tool to indicate that it has loaded/unloaded the shuttle

//IF THIS^.Sealer.sealbar.InTempRange THEN
	ChangeState(E_PMLCommand.ePMLCommand_Unsuspend);
//END_IF
END_METHOD

METHOD PROTECTED Suspending
VAR_INPUT
END_VAR
CASE _CurrentMode OF
    //=================================PRODUCTION MODE==================================
    E_PMLUnitMode.ePMLUnitMode_Production:
		CassetteLoaderEM.ShuttleReady := FALSE; //reset 
		
        IF (CassetteLoaderEM.CurrentState = E_PMLState.ePMLState_Complete OR CassetteLoaderEM.CurrentState = E_PMLState.ePMLState_Idle) THEN
            StateComplete();
        END_IF
    E_PMLUnitMode.ePMLUnitMode_Maintenance, E_PMLUnitMode.ePMLUnitMode_Manual:
        SUPER^.Suspending();
END_CASE
END_METHOD

METHOD PROTECTED Unholding
VAR_INPUT
END_VAR
CASE _CurrentMode OF
    //=================================PRODUCTION MODE==================================
    E_PMLUnitMode.ePMLUnitMode_Production:
        StateComplete();
    E_PMLUnitMode.ePMLUnitMode_Maintenance, E_PMLUnitMode.ePMLUnitMode_Manual:
        SUPER^.Unholding();
END_CASE
END_METHOD

METHOD PROTECTED Unsuspending
VAR_INPUT
END_VAR
CASE _CurrentMode OF
    //=================================PRODUCTION MODE==================================
    E_PMLUnitMode.ePMLUnitMode_Production:
		CassetteLoaderEM.ShuttleReady := TRUE;
        StateComplete();
    E_PMLUnitMode.ePMLUnitMode_Maintenance, E_PMLUnitMode.ePMLUnitMode_Manual:
        SUPER^.Unsuspending();
END_CASE
END_METHOD

METHOD UpdateModeTimers
VAR
    currentTime  : T_DCTIME64;
    timeToUpdate : LREAL;
END_VAR

VAR_INST
    lastTime  : T_DCTIME64 := F_GetActualDcTime64();
    lastState : DINT;
    lastMode  : DINT;
END_VAR
IF _PackTags.Status.StateCurrent <> lastState THEN
    MEMSET(ADR(_PackTags.Admin.StateCurrentTime), 0, SIZEOF(_PackTags.Admin.StateCurrentTime));
    lastState := _PackTags.Status.StateCurrent;
END_IF

IF _PackTags.Status.UnitModeCurrent <> lastMode THEN
    MEMSET(ADR(_PackTags.Admin.ModeCurrentTime), 0, SIZEOF(_PackTags.Admin.ModeCurrentTime));
    lastMode := _PackTags.Status.UnitModeCurrent;
END_IF

currentTime := F_GetActualDcTime64();
IF lastTime <> 0 THEN
    timeToUpdate := ULINT_TO_LREAL(currentTime - lastTime) / 1_000_000_000.0;
END_IF

// only seconds get added to the cumulative timers 
IF timeToUpdate > 1 THEN
    _PackTags.Admin.ModeCummulativeTime[_PackTags.Status.UnitModeCurrent] := _PackTags.Admin.ModeCummulativeTime[_PackTags.Status.UnitModeCurrent] + LREAL_TO_DINT(timeToUpdate);
    _PackTags.Admin.ModeCurrentTime[_PackTags.Status.UnitModeCurrent]     := _PackTags.Admin.ModeCurrentTime[_PackTags.Status.UnitModeCurrent] + LREAL_TO_DINT(timeToUpdate);
    _PackTags.Admin.StateCummulativeTime[_PackTags.Status.UnitModeCurrent, _PackTags.Status.StateCurrent]
        := _PackTags.Admin.StateCummulativeTime[_PackTags.Status.UnitModeCurrent, _PackTags.Status.StateCurrent] + LREAL_TO_DINT(timeToUpdate);

    _PackTags.Admin.StateCurrentTime[_PackTags.Status.UnitModeCurrent, _PackTags.Status.StateCurrent] :=
        _PackTags.Admin.StateCurrentTime[_PackTags.Status.UnitModeCurrent, _PackTags.Status.StateCurrent] + LREAL_TO_DINT(timeToUpdate);

    lastTime := currentTime;
END_IF
END_METHOD

END_FUNCTION_BLOCK

// ---- Machine/EquipmentModules/FB_CassetteLoader.TcPOU
FUNCTION_BLOCK FB_CassetteLoader EXTENDS FB_PackML_BaseModule

VAR
	    // Sub module definitions here

    // List of sub modules
    ipSubModules_Init : ARRAY[1..Parameters_PackML_Base.MAX_NO_OF_SUBMODULES] OF I_PackML_BaseModule := [];

    // Component definitions here
    ElevatorAxisA : FB_Component_BasicAxis := (Name := 'ElevatorA');
	ElevatorAxisB : FB_Component_BasicAxis := (Name := 'ElevatorB');
	ShuttleAxis : FB_Component_BasicAxis := (Name := 'Shuttle');
	MapSensorA : FB_DigitalSensor := (Name := 'MapSensorA');
	MapSensorB : FB_DigitalSensor := (Name := 'MapSensorB');
	
	//Assign Homing Routine to Use the Absolute Encoder, using the persistent struct below
	AbsHomingElevA : FB_HomeRoutine_AbsHoming;
	AbsHomingElevB : FB_HomeRoutine_AbsHoming;
	AbsHomingShuttle : FB_HomeRoutine_AbsHoming;
		
	//Alarms for this Module
	LoaderAlarms : ARRAY[1..LOADER_ALARM_COUNT] OF FB_TcAlarm;
	
	//Data for module
    Recipe : ST_LoaderRecipe;
	CassetteAStatus : ST_CassetteStatus;
	CassetteBStatus : ST_CassetteStatus;
	_ElevatorAxisAStagePosition : LREAL;
	_ElevatorAxisBStagePosition : LREAL;
	_ShuttleAxisStagePosition : LREAL;
	_ElevatorAxisAHomePosition : LREAL;
	_ElevatorAxisBHomePosition : LREAL;
	_ShuttleAxisHomePosition : LREAL;
	
	//HMI Control for EM
    fbControlSourceHMI : FB_ControlSource_HMI;
	
	//Load or Unload Mode: Commanded by External, TRUE= Load, FALSE = Unload
	_LoadOrUnload : BOOL;
	_ShuttleReady : BOOL;

	//This trigger each axis at the abs zero position when in maintenance or manual mode
	AbsHomeCmdA: BOOL;
	AbsHomeCmdB: BOOL;
	AbsHomeCmdShuttle: BOOL;
	_NeedsMapping: BOOL;
	_NextSlot: DINT;
	_NextCassette: INT;
END_VAR

VAR CONSTANT
	LOADER_ALARM_COUNT : INT := 6;
END_VAR

VAR PERSISTENT
	ElevAHomingParameters : ST_AbsHomeParameters;
	ElevBHomingParameters : ST_AbsHomeParameters;
	ShuttleHomingParameters : ST_AbsHomeParameters;
END_VAR

ShuttleHomingParameters.PositionBias := 0;

METHOD PROTECTED Aborting
VAR_INPUT
END_VAR
CASE SequenceState OF
    0:
        NoStateTasksToComplete := FALSE;
        SequenceState          := SequenceState + 10;
    10:
        ElevatorAxisA.Stop();
		ElevatorAxisB.Stop();
		ShuttleAxis.Stop();
//        IF (ElevatorAxisA.Stopped AND ElevatorAxisB.Stopped AND ShuttleAxis.Stopped) THEN
//            SequenceState := SequenceState + 10;
//        END_IF
		SequenceState := SequenceState + 10;
    20:
        // Disable here
        ElevatorAxisA.Disable();
		ElevatorAxisB.Disable();
		ShuttleAxis.Disable();

        // Check not enabled here
        IF NOT (ElevatorAxisA.Enabled AND ElevatorAxisB.Enabled AND ShuttleAxis.Enabled) THEN
            SequenceState := SequenceState + 10;
        END_IF
    30:
        StateTasksComplete := TRUE;
END_CASE

SUPER^.Aborting();
END_METHOD

PROPERTY BladeThickness : LREAL
GET
BladeThickness := recipe.Elevator.BladeThickness;
END_GET
SET
BladeThickness := recipe.Elevator.BladeThickness;
END_SET
END_PROPERTY

PROPERTY CassettePitch : LREAL
GET
CassettePitch := recipe.Elevator.CassettePitch;
END_GET
SET
recipe.Elevator.CassettePitch := CassettePitch;
END_SET
END_PROPERTY

PROPERTY CassetteSlotHeight : LREAL
GET
CassetteSlotHeight := recipe.Elevator.CassetteSlotHeight;
END_GET
SET
recipe.Elevator.CassetteSlotHeight := CassetteSlotHeight;
END_SET
END_PROPERTY

PROPERTY CassetteSlotNumber : INT
GET
CassetteSlotNumber := recipe.Elevator.CassetteSlotNumber;
END_GET
SET
recipe.Elevator.CassetteSlotNumber := CassetteSlotNumber;
END_SET
END_PROPERTY

METHOD PROTECTED Clearing
VAR_INPUT
END_VAR
CASE SequenceState OF
    0:
        NoStateTasksToComplete := FALSE;
        SequenceState          := SequenceState + 10;
	10:
        //Reset any alarms that get latched
        //PullWheelAlarms[E_PullWheels.StartTimeout].Clear(0, 0);
        SequenceState := SequenceState + 10;
    20:
        StateTasksComplete := TRUE;
END_CASE

SUPER^.Clearing();
END_METHOD

METHOD CyclicLogic
VAR_INPUT
END_VAR

VAR
	i : INT;
	TotalInCassetteA : INT;
	TotalInCassetteB : INT;
	CassetteAInteger : ARRAY[0..23] OF INT; //matching array with INT type
	CassetteBInteger : ARRAY[0..23] OF INT; //matching array with INT type
END_VAR
IF NOT _InitComplete THEN
    _InitComplete := Initialize();
    RETURN;
END_IF

SUPER^.CyclicLogic();

//Set the current alarm severity for this module
_CurrentAlarmSeverity   := F_GetMaxSeverityRaised(Alarms := LoaderAlarms, CurrentSeverity := _CurrentAlarmSeverity);

//Add up the number of waveguides in each cassette and mark the cassette status as full
	FOR i := 0 TO 23 DO
		IF CassetteAStatus.WaveguidePresent[i] = TRUE THEN
			CassetteAInteger[i] := 1;
		ELSE
			CassetteAInteger[i] := 0;
		END_IF
		TotalInCassetteA := TotalInCassetteA + CassetteAInteger[i];
		IF TotalInCassetteA > 22 THEN
			CassetteAStatus.CassetteFull := TRUE;
		END_IF
	END_FOR; 
	
	FOR i := 0 TO 23 DO
		IF CassetteBStatus.WaveguidePresent[i] = TRUE THEN
			CassetteBInteger[i] := 1;
		ELSE
			CassetteBInteger[i] := 0;
		END_IF
		TotalInCassetteB := TotalInCassetteB + CassetteBInteger[i];
		IF TotalInCassetteB > 22 THEN
			CassetteBStatus.CassetteFull := TRUE;
		END_IF
	END_FOR;
END_METHOD

METHOD DetermineNextSlot : DINT
VAR_INPUT
	CassetteID : ST_CassetteStatus;
END_VAR

VAR
	i: DINT;
END_VAR
//This method searches the wafer map array from the bottom to the top, returning the highest slot that is empty
	FOR i := 0 TO 23 DO
		IF CassetteID.WaveguidePresent[i] = FALSE THEN
			DetermineNextSlot := i;
		END_IF
	END_FOR;
END_METHOD

METHOD DetermineNextWaveguide : INT
VAR_INPUT
		CassetteID : ST_CassetteStatus;
END_VAR

VAR
	i: INT;
END_VAR
//This method searches the wafer map array from the bottom to the top, returning the lowest slot that is full
	FOR i := 23 TO 0 DO
		IF CassetteID.WaveguidePresent[i] = TRUE THEN
			DetermineNextWaveguide := i;
		END_IF
	END_FOR;
END_METHOD

PROPERTY ElevatorAcceleration : LREAL
GET
ElevatorAcceleration := recipe.Elevator.Acceleration;
END_GET
SET
recipe.Elevator.Acceleration := ElevatorAcceleration;
END_SET
END_PROPERTY

PROPERTY ElevatorFirstWaveguidePosition : LREAL
GET
ElevatorFirstWaveguidePosition := recipe.Elevator.FirstWaveguidePosition;
END_GET
SET
recipe.Elevator.FirstWaveguidePosition := ElevatorFirstWaveguidePosition;
END_SET
END_PROPERTY

PROPERTY ElevatorVelocity : LREAL
GET
ElevatorVelocity := recipe.Elevator.Velocity;
END_GET
SET
recipe.Elevator.Velocity := ElevatorVelocity;
END_SET
END_PROPERTY

METHOD PROTECTED Execute
VAR_INPUT
END_VAR
CASE _CurrentMode OF
    //=================================PRODUCTION MODE==================================
    E_PMLUnitMode.ePMLUnitMode_Production:
		IF _LoadOrUnload = TRUE THEN // _LoadOrUnload = TRUE means LOAD the cassette
			
		//Loading case
			CASE SequenceState OF

				10:		//Figure out where to put the next waveguide
						//we will load cassette A (top-down) before cassette B (top-down), so if A is full start loading B 
						IF NOT CassetteAStatus.CassetteFull THEN
							_NextSlot := DetermineNextSlot(CassetteID := CassetteAStatus);
							_NextCassette := 0; 
						ELSE	
							_NextSlot := DetermineNextSlot(CassetteID := CassetteBStatus);
							_NextCassette := 1;
						END_IF
						SequenceState := SequenceState + 10;
				20:		//Make sure that the space under/over the slot is clear, abort if obstructed
						IF _NextCassette = 0 THEN
							IF (CassetteAStatus.ClearBelowWaveguide[_NextSlot] AND CassetteAStatus.ClearBelowWaveguide[_NextSlot + 1]) = TRUE THEN
								SequenceState := SequenceState + 10;
							ELSE
								//changestate(ePMLState_Aborting);
							END_IF
						ELSE
							IF (CassetteBStatus.ClearBelowWaveguide[_NextSlot] AND CassetteBStatus.ClearBelowWaveguide[_NextSlot + 1]) = TRUE THEN
								SequenceState := SequenceState + 10;
							ELSE
								//changestate(ePMLState_Aborting);
							END_IF
						END_IF
						SequenceState := SequenceState + 10;
				30: 	//Move all to staged position
						SequenceState := SequenceState + 10;
				40:		//Call PlaceToNextOpenSlot method
						PlaceToNextOpenSlot(_NextCassette, _NextSlot);
						SequenceState := SequenceState + 10;
				50:		//Depending on which cassette we loaded, update the map to add the waveguide:
						IF _NextCassette = 0 THEN
							CassetteAStatus.WaveguidePresent[_NextSlot]:= 1;
						ELSE
							CassetteBStatus.WaveguidePresent[_NextSlot]:= 1;
						END_IF
						SequenceState := SequenceState + 10;

				99:		//based on the cassette status, either go into suspending or completing
						IF (CassetteAStatus.CassetteFull AND CassetteBStatus.CassetteFull) THEN
							StateComplete();
						ELSE
							//go into suspending state
							//changestate(ePMLState_Suspending);
						END_IF
			END_CASE
			
		//Unload Case	
		ELSE //_LoadOrUnload = FALSE means UNLOAD the cassette
			
			CASE SequenceState OF
				10: //Figure out which waveguide to remove first
				//we will unload cassette A (bottom-up) before cassette B (bottom-up), so if A is empty start unloading B
						IF CassetteAStatus.CassetteFull THEN
							_NextSlot := DetermineNextWaveguide(CassetteID := CassetteAStatus);
							_NextCassette := 0; 
						ELSE	
							_NextSlot := DetermineNextWaveguide(CassetteID := CassetteBStatus);
							_NextCassette := 1;
						END_IF
						SequenceState := SequenceState + 10;
				20:		//Make sure that the space under/over the slot is clear, abort if obstructed
						IF _NextCassette = 0 THEN
							IF (CassetteAStatus.ClearBelowWaveguide[_NextSlot] AND CassetteAStatus.ClearBelowWaveguide[_NextSlot + 1]) = TRUE THEN
								SequenceState := SequenceState + 10;
							ELSE
								//changestate(ePMLState_Aborting);
							END_IF
						ELSE
							IF (CassetteBStatus.ClearBelowWaveguide[_NextSlot] AND CassetteBStatus.ClearBelowWaveguide[_NextSlot + 1]) = TRUE THEN
								SequenceState := SequenceState + 10;
							ELSE
								//changestate(ePMLState_Aborting);
							END_IF
						END_IF
						SequenceState := SequenceState + 10;
				30:		//Pre-position the stages
						IF _NextCassette = 0 THEN
							ElevatorAxisA.MoveAbsolute(_ElevatorAxisAStagePosition,TRUE);
							ElevatorAxisB.MoveAbsolute(_ElevatorAxisBHomePosition,TRUE);
							ShuttleAxis.MoveAbsolute(_ShuttleAxisStagePosition, TRUE);
						ELSE
							ElevatorAxisA.MoveAbsolute(_ElevatorAxisAHomePosition,TRUE);
							ElevatorAxisB.MoveAbsolute(_ElevatorAxisBStagePosition,TRUE);
							ShuttleAxis.MoveAbsolute(_ShuttleAxisStagePosition, TRUE);
						END_IF
						SequenceState := SequenceState + 10;
				40: 	//Confirm all axis preposition movements are complete
						IF (ElevatorAxisA.Busy AND ElevatorAxisB.Busy AND ShuttleAxis.Busy) THEN
							SequenceState := SequenceState + 10;
						END_IF
				50:		//Call GetNextWaveguide method
						GetNextWaveGuide(_NextCassette, _NextSlot);
						SequenceState := SequenceState + 10;
				60:		//Depending on which cassette we unloaded, update the map to remove the waveguide:
						IF _NextCassette = 0 THEN
							CassetteAStatus.WaveguidePresent[_NextSlot]:= 0;
						ELSE
							CassetteBStatus.WaveguidePresent[_NextSlot]:= 0;
						END_IF
						SequenceState := SequenceState + 10;
				
			END_CASE
		END_IF
//If we are waiting for the tool to load/unload the waveguide, switch to Suspending state



    //=================================MAINTENANCE & MANUAL MODE==================================		
    E_PMLUnitMode.ePMLUnitMode_Maintenance, E_PMLUnitMode.ePMLUnitMode_Manual:
        //Reset the abs zero position when commanded
		IF AbsHomeCmdA THEN
    		AbsHomingElevA.Execute();
    		AbsHomeCmdA:=FALSE;
		END_IF;
		
		IF AbsHomeCmdB THEN
    		AbsHomingElevA.Execute();
    		AbsHomeCmdB:=FALSE;
		END_IF;
		
		IF AbsHomeCmdShuttle THEN
    		AbsHomingElevA.Execute();
    		AbsHomeCmdShuttle:=FALSE;
		END_IF;
END_CASE
END_METHOD

METHOD GetNextWaveguide : BOOL
VAR_INPUT
	NextCassette : INT;
	NextSlot : DINT;
END_VAR
//This method will get the waveguide in the cassette and slot defined as next-available and move the shuttle to the tool position
END_METHOD

//! @summary Basic module initialization logic
METHOD PROTECTED Initialize : BOOL;
VAR
	i						 : UDINT;
	varInfo					 : __SYSTEM.VAR_INFO;
	AllSubUnitsInitialized	 : BOOL := TRUE;
	AllComponentsInitialized : BOOL := TRUE;
END_VAR

//! @description This method is called by <c>CyclicLogic()</c> as required
Initialize := FALSE;
CASE DescendantSequenceState OF
    0:
		//RegisterComponent here (none for now)
        _LogModeChanges         := FALSE;
        _LogStateChanges        := FALSE;
        DescendantSequenceState := DescendantSequenceState + 10;
    10:
        //Setup Custom modes here
        CustomModes(eMode                          :=,
                    sName                          := 'Name',
                    bDisableClearing               := FALSE,
                    bDisableStarting               := FALSE,
                    bDisableSuspended              := FALSE,
                    bDisableStopping               := FALSE,
                    bDisableAborting               := FALSE,
                    bDisableHolding                := TRUE, //no operator hold state 
                    bDisableHeld                   := TRUE,
                    bDisableUnholding              := TRUE,
                    bDisableSuspending             := FALSE,
                    bDisableUnsuspending           := FALSE,
                    bDisableResetting              := FALSE,
                    bDisableIdle                   := FALSE,
                    bDisableCompleting             := FALSE,
                    bDisableComplete               := FALSE,
                    bEnableUnitModeChangeStopped   := TRUE,
                    bEnableUnitModeChangeIdle      := TRUE,
                    bEnableUnitModeChangeSuspended := FALSE,
                    bEnableUnitModeChangeExecute   := FALSE,
                    bEnableUnitModeChangeAborted   := FALSE,
                    bEnableUnitModeChangeHeld      := FALSE,
                    bEnableUnitModeChangeComplete  := FALSE,
                    bError                         =>,
                    nErrorId                       =>);
        DescendantSequenceState := DescendantSequenceState + 10;
    20:
        //Copy Mode names
        FOR i := 1 TO 3 DO
            ModeNames[i] := F_UnitModeToString(UDINT_TO_DINT(i));
        END_FOR

        //Initialize_TagData();
		RegisterExternalController(Controller := fbControlSourceHMI);
		fbControlSourceHMI.CyclicLogic();
        DescendantSequenceState := DescendantSequenceState + 10;
		
	30: //Register homing methods for each axis
//				ShuttleAxis.HomeMethod := AbsHomingShuttle;
//				AbsHomingShuttle.Parameters := ShuttleHomingParameters;
//				ElevatorAxisA.HomeMethod := AbsHomingElevA;
//				AbsHomingElevA.Parameters := ElevAHomingParameters;
//				ElevatorAxisB.HomeMethod := AbsHomingElevB;
//				AbsHomingElevB.Parameters := ElevBHomingParameters;
      	DescendantSequenceState := DescendantSequenceState + 10;
    40:
        //Call the Super
        IF SUPER^.Initialize() THEN
            DescendantSequenceState := DescendantSequenceState + 10;
        END_IF
    50:
        Initialize := TRUE;
END_CASE
END_METHOD

METHOD LoadCassette : BOOL
VAR_INPUT

END_VAR
(* This method will allow the user to stop the machine, open the door, install cassettes, 
close the door, restart the machine, map the cassettes and go into a ready state *)
END_METHOD

PROPERTY LoadOrUnload : bool
GET
LoadOrUnload := _LoadOrUnload;
END_GET
SET
_LoadOrUnload := LoadOrUnload;
END_SET
END_PROPERTY

METHOD MapCassette : BOOL
VAR_INPUT
	CassetteToMap : INT; //Cassette A is zero, Cassette B is one, etc.
END_VAR

VAR
	
END_VAR

//this method will map the cassette specified in CassetteToMap, saving the output in the array CassetteAStatus.WaveguidePresent
END_METHOD

METHOD PlaceToNextOpenSlot : BOOL
VAR_INPUT
	NextCassette : INT;
	NextSlot : DINT;
END_VAR
//This method will place the waveguide (placed on the blade by the tool) to the next open slot
END_METHOD

METHOD PROTECTED Resetting
VAR_INPUT
END_VAR
CASE _CurrentMode OF
    //=================================PRODUCTION MODE==================================
    E_PMLUnitMode.ePMLUnitMode_Production:
        CASE SequenceState OF
            0:
                NoStateTasksToComplete := FALSE;
                SequenceState          := SequenceState + 10;
            10:
				// Enable here
				ElevatorAxisA.Enable();
				ElevatorAxisB.Enable();
				ShuttleAxis.Enable();	
				// Check enabled here
				IF (ElevatorAxisA.Enabled AND ElevatorAxisB.Enabled AND ShuttleAxis.Enabled) THEN
					StateTasksComplete := TRUE;
				END_IF
                //SequenceState := SequenceState + 10;
            20:
                //IF (*LeftPullWheel.InGear AND*) RightPullWheel.InGear THEN
                    //StateTasksComplete := TRUE;
                //END_IF
        END_CASE

    //=================================MAINTENANCE & MANUAL MODE==================================	
    E_PMLUnitMode.ePMLUnitMode_Maintenance, E_PMLUnitMode.ePMLUnitMode_Manual:
        ;
END_CASE

SUPER^.Resetting();
END_METHOD

PROPERTY ShuttleCassettePosition : LREAL
GET
ShuttleCassettePosition := recipe.Shuttle.CassettePosition;
END_GET
SET
recipe.Shuttle.CassettePosition := ShuttleCassettePosition;
END_SET
END_PROPERTY

PROPERTY ShuttleReady : BOOL
GET
ShuttleReady := _ShuttleReady;
END_GET
SET
_ShuttleReady := ShuttleReady;
END_SET
END_PROPERTY

PROPERTY ShuttleToolPosition : LREAL
GET
ShuttleToolPosition := recipe.Shuttle.ToolPosition;
END_GET
SET
recipe.Shuttle.ToolPosition := ShuttleToolPosition;
END_SET
END_PROPERTY

PROPERTY ShuttleVelocity : LREAL
GET
ShuttleVelocity := recipe.Shuttle.Velocity;
END_GET
SET
recipe.Shuttle.Velocity := ShuttleVelocity;
END_SET
END_PROPERTY

//! @summary This method contains code which will execute when this PackML module is in the <b>Starting</b> state
METHOD PROTECTED Starting
VAR
	i				: UDINT;
	SubModulesReady : BOOL := TRUE;
END_VAR

(*! <description><b></b><table> 
	<tr>
		<th> Previous State </th>
		<th> Transition In </th>
		<th> Transition Out </th>
		<th> Next State  </th> 
	</tr>
	<tr>
		<td> Idle </td>
		<td> Start Command </td> 
		<td> State Complete </td>
		<td> Execute </td> 
	</tr>
</table>
This method is called as required by <c>StateControl()</c>
</description> 

*)
CASE _CurrentMode OF
    //=================================PRODUCTION MODE==================================
    E_PMLUnitMode.ePMLUnitMode_Production:
        CASE SequenceState OF
            0:
                NoStateTasksToComplete := FALSE;
                SequenceState          := SequenceState + 10;
            10:
                //assign all recipe values here
				ElevatorAxisA.Velocity := Recipe.Elevator.Velocity;
				ElevatorAxisA.Acceleration := Recipe.Elevator.Acceleration;
                SequenceState := SequenceState + 10;
			20:
				//Home the shuttle axis
				ShuttleAxis.Home();
				SequenceState := SequenceState + 10;
			30: 
				//Home the elevator axis at the same time
				ElevatorAxisA.Home();
				ElevatorAxisB.Home();
				SequenceState := SequenceState + 10;
			40: //With the elevator stages at home, map each cassette
				MapCassette(0);
				IF NOT ElevatorAxisA.Busy THEN
					SequenceState := SequenceState + 10;
				END_IF
			50: //
				MapCassette(1);
				IF NOT ElevatorAxisB.Busy THEN
					SequenceState := SequenceState + 10;
				END_IF
            60:
				//Verify that home is completed and home sensors are satisfied
                IF NOT (ElevatorAxisA.Busy AND ElevatorAxisB.Busy AND ShuttleAxis.Busy) THEN
                    StateTasksComplete := TRUE;
                END_IF
        END_CASE

    //=================================MAINTENANCE & MANUAL MODE==================================
    E_PMLUnitMode.ePMLUnitMode_Maintenance, E_PMLUnitMode.ePMLUnitMode_Manual:
        ;
END_CASE
END_METHOD

METHOD PROTECTED Stopping
VAR_INPUT
END_VAR
CASE _CurrentMode OF
    //=================================PRODUCTION MODE==================================
	//	The elevators and shuttle are disabled, so they can not be moved. Does this state do anything?
	
    E_PMLUnitMode.ePMLUnitMode_Production:
        CASE SequenceState OF
            0:
                NoStateTasksToComplete := FALSE;
                //PullWheelCylinder.Retract();
                SequenceState := SequenceState + 10;
            10:
				
//                IF PullWheelCylinder.Retracted THEN
//                    SequenceState := SequenceState + 10;
//                END_IF
				SequenceState := SequenceState + 10;
            20:
                StateTasksComplete := TRUE;
        END_CASE

    //=================================MAINTENANCE & MANUAL MODE==================================
    E_PMLUnitMode.ePMLUnitMode_Maintenance, E_PMLUnitMode.ePMLUnitMode_Manual:
        ;
END_CASE

SUPER^.Stopping();
END_METHOD

//! @summary This method contains code which will execute when this PackML module is in the <b>Suspending</b> state
METHOD PROTECTED Suspending
VAR
	i				: UDINT;
	SubModulesReady : BOOL := TRUE;
END_VAR

(*! <description><b>Note:</b> The <i>Suspend</i> command is intended to be initiated by automatic detection of upstream/downstream jams, etc. It is meant to be distinct from a <i>Hold</i> in that <i>Hold</i> should be commanded by an operator.  Both <i>Hold</i>and<i>Suspend</i> result in a <i>paused</i> state which should allow resumption of the <b>Execute</b> state. 
<table> 
	<tr>
		<th> Previous State </th>
		<th> Transition In </th>
		<th> Transition Out </th>
		<th> Next State  </th> 
	</tr>
	<tr>
		<td> Execute </td>
		<td> Suspend Command </td> 
		<td> State Complete </td>
		<td> Suspended </td> 
	</tr>
</table>
This method is called as required by <c>StateControl()</c>
</description> 

*)
//Notify the tool that the shuttle is waiting
END_METHOD

METHOD UnloadCassette : BOOL
VAR_INPUT
END_VAR
(* This method will allow the user to trigger an unload sequence, open the door, remove the cassettes,
close the door and wait for new cassettes *)
END_METHOD

PROPERTY WaveguideThickness : LREAL
GET
WaveguideThickness := recipe.Elevator.WaveguideThickness;
END_GET
SET
recipe.Elevator.WaveguideThickness := WaveguideThickness;
END_SET
END_PROPERTY

END_FUNCTION_BLOCK

// ---- Machine/Templates/FB_EquipmentModuleTemplate.TcPOU
FUNCTION_BLOCK ABSTRACT FB_EquipmentModuleTemplate EXTENDS FB_PackML_BaseModule
VAR
    // Sub module definitions here

    // List of sub modules
    ipSubModules_Init : ARRAY[1..Parameters_PackML_Base.MAX_NO_OF_SUBMODULES] OF I_PackML_BaseModule := [];

    // Component definitions here

    // List of Components
    ipComponents_Init : ARRAY[1..Parameters_PackML_Base.MAX_NO_OF_COMPONENTS] OF I_ComponentBase := [];

    //Parameters from PackTags for module
    _Param : ARRAY[1..10] OF ST_Descriptor2;
END_VAR

METHOD PROTECTED CreateEvents
VAR_INPUT
END_VAR
// Add your event creation here

// Super call to base
SUPER^.CreateEvents();
END_METHOD

METHOD CyclicLogic
VAR_INPUT
END_VAR
IF NOT _InitComplete THEN
    _InitComplete := Initialize();
    RETURN;
END_IF

SUPER^.CyclicLogic();
END_METHOD

//! @summary Basic module initialization logic
METHOD PROTECTED Initialize : BOOL;
VAR
    i                        : UDINT;
    varInfo                  : __SYSTEM.VAR_INFO;
    AllSubUnitsInitialized   : BOOL := TRUE;
    AllComponentsInitialized : BOOL := TRUE;
END_VAR

//! @description This method is called by <c>CyclicLogic()</c> as required
Initialize := FALSE;
CASE DescendantSequenceState OF
    0:
        // Define the interfaces to the different subunits (Must take place before SUPER^.initialize call)
        FOR i := 1 TO SPT_PackMLBase.Parameters_PackML_Base.MAX_NO_OF_SUBMODULES DO
            ipSubModules[i] := ipSubModules_Init[i];
        END_FOR

        FOR i := 1 TO SPT_PackMLBase.Parameters_PackML_Base.MAX_NO_OF_COMPONENTS DO
            ipComponents[i] := ipComponents_Init[i];
        END_FOR

        _LogModeChanges         := FALSE;
        _LogStateChanges        := FALSE;
        DescendantSequenceState := DescendantSequenceState + 10;
    10:
        //Setup Custom modes here

        (*CustomModes(eMode                          :=,
                    sName                          :=,
                    bDisableClearing               :=,
                    bDisableStarting               :=,
                    bDisableSuspended              :=,
                    bDisableStopping               :=,
                    bDisableAborting               :=,
                    bDisableHolding                :=,
                    bDisableHeld                   :=,
                    bDisableUnholding              :=,
                    bDisableSuspending             :=,
                    bDisableUnsuspending           :=,
                    bDisableResetting              :=,
                    bDisableIdle                   :=,
                    bDisableCompleting             :=,
                    bDisableComplete               :=,
                    bEnableUnitModeChangeStopped   :=,
                    bEnableUnitModeChangeIdle      :=,
                    bEnableUnitModeChangeSuspended :=,
                    bEnableUnitModeChangeExecute   :=,
                    bEnableUnitModeChangeAborted   :=,
                    bEnableUnitModeChangeHeld      :=,
                    bEnableUnitModeChangeComplete  :=,
                    bError                         =>,
                    nErrorId                       =>);*)
        DescendantSequenceState := DescendantSequenceState + 10;
    20:
        //Copy Mode names
        DescendantSequenceState := DescendantSequenceState + 10;
    30:
        //Call the Super
        IF SUPER^.Initialize() THEN
            DescendantSequenceState := DescendantSequenceState + 10;
        END_IF
    40:
        Initialize := TRUE;
END_CASE
END_METHOD

METHOD RaiseAlarm2Args
VAR_IN_OUT
    fbAlarm : FB_TcAlarm; //Alarm to be raised
END_VAR

VAR_INPUT
    String_1 : STRING; //First String Parameter (The Name of this component will be applied first automatically)
    String_2 : STRING; //Second String Parameter
END_VAR
F_RaiseAlarmWithStringParameters(Alarm    := fbAlarm,
                                 String_1 := Name,
                                 String_2 := String_1,
                                 String_3 := String_2);
END_METHOD

METHOD SetParam
VAR_INPUT
    ParamID   : DINT;
    Parameter : ST_Descriptor2;
END_VAR
_Param[ParamID] := Parameter;
END_METHOD

END_FUNCTION_BLOCK

// ---- GlobalTextList.TcGTLO
TEXTLIST GlobalTextList
  733 = '%0.1f °'
  685 = '%s'
  680 = 'Abort'
  452 = 'Clear'
  809 = 'Clear Unwind'
  9 = 'Clear Unwinder'
  504 = 'Command'
  424 = 'EStop'
  744 = 'Hold'
  324 = 'Load / Unload Complete'
  618 = 'Loading Mode'
  517 = 'Low Air'
  347 = 'MACHINE'
  46 = 'Maintenance'
  904 = 'Manual'
  929 = 'Production'
  181 = 'Reset'
  538 = 'Reset Unwind'
  902 = 'Shuttle Ready'
  77 = 'Start'
  804 = 'Start Unwind'
  516 = 'State: %s'
  828 = 'Stop'
  806 = 'Suspend'
  995 = 'Temp Setpoint'
  197 = 'Unhold'
  196 = 'Unloading Mode'
  832 = 'Unsuspend'
  702 = 'Unsuspend / Get Next'
END_TEXTLIST

// ---- VISUs/VisuOjects/V_MachineModule.TcVIS
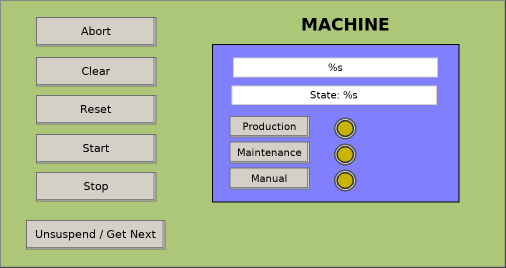
VISUALIZATION V_MachineModule  // 506x268
VAR_IN_OUT
	HMI : ST_PackMLModuleBase_HMI;
END_VAR
    RoundedRectangle (0,0 506x268)
    Button (36,17 120x29), "Abort"
        OnMouseClick: execute { HMI.Command.State := E_PMLCommand.ePMLCommand_Abort; }
    Button (36,57 120x29), "Clear"
        OnMouseClick: execute { HMI.Command.State := E_PMLCommand.ePMLCommand_Clear; }
    Button (36,95 120x29), "Reset"
        OnMouseClick: execute { HMI.Command.State := E_PMLCommand.ePMLCommand_Reset; }
    Button (36,134 120x29), "Start"
        OnMouseClick: execute { HMI.Command.State := E_PMLCommand.ePMLCommand_Start; }
    Button (36,172 120x29), "Stop"
        OnMouseClick: execute { HMI.Command.State := E_PMLCommand.ePMLCommand_Stop; }
    Button (26,220 139x29), "Unsuspend / Get Next"
        OnMouseClick: execute { HMI.Command.State := E_PMLCommand.ePMLCommand_Unsuspend; }
    Frame (212,44 247x158)
        shows V_Module(HMI := HMI)
    Label (229,6 233x37), "MACHINE"
END_VISUALIZATION

// ---- VISUs/VisuOjects/V_Module.TcVIS
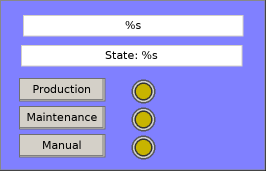
VISUALIZATION V_Module  // 266x171
VAR_IN_OUT
	HMI : ST_PackMLBaseModule_HMI;
END_VAR
    RoundedRectangle (0,0 266x171)
    Textfield (23,15 220x21), "%s", text variable: HMI.Config.Name
    Textfield (21,45 221x21), "State: %s", text variable: HMI.Status.State
    Button (19,78 86x23), "Production"
        OnMouseClick: execute { HMI.Command.Mode := E_PMLUnitMode.ePMLUnitMode_Production; }
    Button (19,106 86x23), "Maintenance"
        OnMouseClick: execute { HMI.Command.Mode := E_PMLUnitMode.ePMLUnitMode_Maintenance; }
    Button (19,134 86x23), "Manual"
        OnMouseClick: execute { HMI.Command.Mode := E_PMLUnitMode.ePMLUnitMode_Manual; }
    Lamp1 (130,78 27x27), variable: HMI.Status.Mode = E_PMLUnitMode.ePMLUnitMode_Production, style: Lamp-Lamp1-Yellow
    Lamp1 (130,106 27x27), variable: HMI.Status.Mode = E_PMLUnitMode.ePMLUnitMode_Maintenance, style: Lamp-Lamp1-Yellow
    Lamp1 (130,134 27x27), variable: HMI.Status.Mode = E_PMLUnitMode.ePMLUnitMode_Manual, style: Lamp-Lamp1-Yellow
END_VISUALIZATION

// ---- VISUs/V_Main.TcVIS
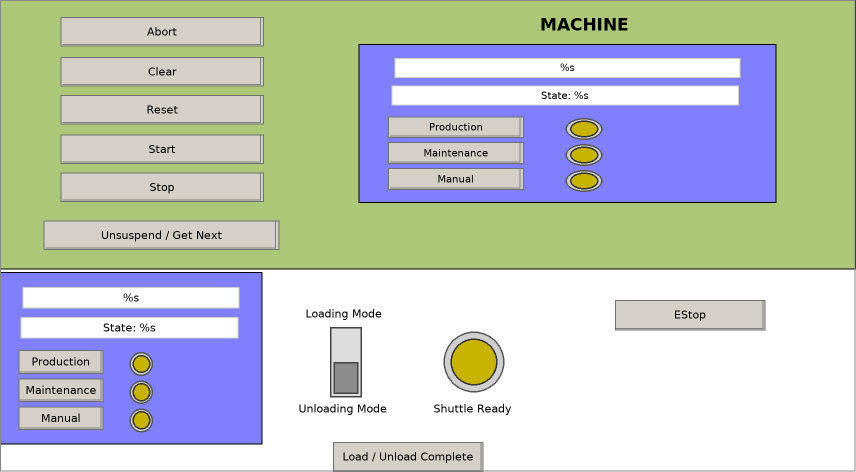
VISUALIZATION V_Main  // 856x472
    Frame (0,0 856x269)
        shows V_MachineModule(HMI := MAIN.CassetteLoaderMachine.PackMLBaseModule_HMI)
    Frame (0,272 262x172)
        shows V_Module(HMI := MAIN.CassetteLoaderMachine.CassetteLoaderEM.PackMLBaseModule_HMI)
    Button (615,300 150x30), "EStop"
        toggle MAIN.CassetteLoaderMachine.EstopInput
    Button (333,442 150x30), "Load / Unload Complete"
        toggle MAIN.CassetteLoaderMachine.LowAirInput
    DipSwitch (311,327 70x70), variable: MAIN.CassetteLoaderMachine.CassetteLoaderEM._LoadOrUnload, behaviour: TOGGLE, style: Switch-DipSwitch-Gray
    Label (269,299 150x30), "Loading Mode"
    Label (268,394 150x30), "Unloading Mode"
    Lamp1 (439,327 70x70), style: Lamp-Lamp1-Yellow
    Label (424,394 97x30), "Shuttle Ready"
END_VISUALIZATION
